C07243=1098.662,-38.451,-51.109,175.839,14.476,151.944
C07244=1098.667,-38.202,-51.121,175.841,14.477,151.943
C07245=1098.673,-37.951,-51.133,175.843,14.477,151.943
C07246=1098.679,-37.701,-51.145,175.845,14.478,151.943
C07247=1098.684,-37.452,-51.157,175.847,14.478,151.942
C07248=1098.691,-37.202,-51.169,175.849,14.479,151.942
C07249=1098.697,-36.953,-51.182,175.851,14.480,151.942
C07250=1098.702,-36.703,-51.194,175.852,14.481,151.942
C07251=1098.708,-36.453,-51.207,175.854,14.481,151.941
C07252=1098.714,-36.204,-51.219,175.856,14.482,151.941
C07253=1098.720,-35.955,-51.231,175.858,14.482,151.941
C07254=1098.726,-35.705,-51.243,175.859,14.483,151.940
C07255=1098.732,-35.455,-51.256,175.861,14.483,151.940
C07256=1098.738,-35.205,-51.269,175.863,14.484,151.940
C07257=1098.743,-34.956,-51.281,175.865,14.485,151.940
C07258=1098.749,-34.706,-51.293,175.867,14.486,151.939
C07259=1098.755,-34.456,-51.305,175.869,14.486,151.939
C07260=1098.761,-34.207,-51.317,175.871,14.487,151.939
C07261=1098.767,-33.957,-51.330,175.873,14.487,151.938
C07262=1098.773,-33.707,-51.343,175.875,14.488,151.938
C07263=1098.778,-33.458,-51.355,175.877,14.489,151.938
C07264=1098.784,-33.208,-51.367,175.879,14.490,151.938
C07265=1098.790,-32.959,-51.380,175.880,14.490,151.937
C07266=1098.797,-32.692,-51.393,175.883,14.491,151.937
C07267=1098.803,-32.424,-51.407,175.885,14.492,151.937
C07268=1098.809,-32.158,-51.419,175.887,14.493,151.936
C07269=1098.815,-31.891,-51.433,175.889,14.494,151.936
C07270=1098.821,-31.641,-51.446,175.891,14.494,151.936
C07271=1098.827,-31.391,-51.458,175.893,14.495,151.935
C07272=1098.832,-31.142,-51.471,175.895,14.495,151.935
C07273=1098.838,-30.892,-51.483,175.897,14.496,151.935
C07274=1098.845,-30.642,-51.495,175.899,14.497,151.935
C07275=1098.851,-30.392,-51.508,175.901,14.497,151.934
C07276=1098.857,-30.142,-51.520,175.903,14.498,151.934
C07277=1098.862,-29.893,-51.532,175.905,14.499,151.934
C07278=1098.868,-29.644,-51.546,175.907,14.499,151.933
C07279=1098.874,-29.394,-51.558,175.908,14.500,151.933
C07280=1098.880,-29.144,-51.571,175.911,14.500,151.933
C07281=1098.886,-28.894,-51.583,175.912,14.501,151.932
C07282=1098.891,-28.645,-51.595,175.914,14.502,151.932
C07283=1098.897,-28.395,-51.608,175.916,14.503,151.932
C07284=1098.903,-28.146,-51.621,175.918,14.503,151.932
C07285=1098.909,-27.896,-51.634,175.920,14.504,151.931
C07286=1098.916,-27.647,-51.646,175.922,14.504,151.931
C07287=1098.921,-27.397,-51.658,175.924,14.505,151.931
C07288=1098.928,-27.148,-51.671,175.926,14.506,151.930
C07289=1098.933,-26.898,-51.684,175.928,14.507,151.930
C07290=1098.939,-26.648,-51.696,175.930,14.507,151.930
C07291=1098.945,-26.398,-51.709,175.932,14.508,151.930
C07292=1098.950,-26.149,-51.722,175.934,14.509,151.929
C07293=1098.956,-25.900,-51.735,175.936,14.509,151.929
C07294=1098.962,-25.650,-51.748,175.937,14.510,151.929
C07295=1098.968,-25.400,-51.760,175.939,14.511,151.928
C07296=1098.974,-25.150,-51.773,175.942,14.511,151.928
C07297=1098.979,-24.902,-51.786,175.943,14.512,151.928
C07298=1098.985,-24.652,-51.798,175.945,14.513,151.928
C07299=1098.991,-24.402,-51.811,175.947,14.513,151.927
C07300=1098.997,-24.152,-51.824,175.949,14.514,151.927
C07301=1099.003,-23.902,-51.837,175.951,14.515,151.927
C07302=1099.008,-23.652,-51.850,175.953,14.515,151.926
C07303=1099.014,-23.404,-51.862,175.956,14.517,151.926
C07304=1099.020,-23.154,-51.875,175.958,14.517,151.926
C07305=1099.026,-22.904,-51.888,175.960,14.518,151.926
C07306=1099.032,-22.655,-51.901,175.961,14.519,151.925
C07307=1099.038,-22.405,-51.913,175.964,14.519,151.925
C07308=1099.044,-22.155,-51.926,175.965,14.520,151.925
C07309=1099.049,-21.906,-51.939,175.967,14.521,151.924
C07310=1099.055,-21.656,-51.952,175.969,14.521,151.924
C07311=1099.061,-21.406,-51.965,175.971,14.522,151.924
C07312=1099.067,-21.157,-51.978,175.973,14.522,151.923
C07313=1099.073,-20.907,-51.990,175.975,14.523,151.923
C07314=1099.079,-20.658,-52.004,175.977,14.524,151.923
C07315=1099.085,-20.408,-52.016,175.979,14.525,151.923
C07316=1099.090,-20.158,-52.029,175.981,14.525,151.922
C07317=1099.096,-19.909,-52.043,175.983,14.526,151.922
C07318=1099.102,-19.659,-52.055,175.985,14.527,151.922
C07319=1099.108,-19.410,-52.068,175.987,14.527,151.921
C07320=1099.114,-19.160,-52.081,175.989,14.528,151.921
C07321=1099.119,-18.911,-52.095,175.991,14.528,151.921
C07322=1099.125,-18.661,-52.107,175.993,14.529,151.920
C07323=1099.131,-18.412,-52.120,175.995,14.530,151.920
C07324=1099.137,-18.162,-52.133,175.997,14.531,151.920
C07325=1099.143,-17.912,-52.145,175.999,14.531,151.919
C07326=1099.149,-17.662,-52.159,176.001,14.532,151.919
C07327=1099.154,-17.412,-52.172,176.003,14.533,151.919
C07328=1099.161,-17.163,-52.185,176.005,14.534,151.919
C07329=1099.167,-16.914,-52.198,176.007,14.534,151.918
C07330=1099.173,-16.646,-52.211,176.009,14.535,151.918
C07331=1099.179,-16.378,-52.226,176.011,14.536,151.918
C07332=1099.185,-16.110,-52.240,176.014,14.536,151.917
C07333=1099.192,-15.842,-52.254,176.016,14.537,151.917
C07334=1099.198,-15.593,-52.267,176.018,14.538,151.917
C07335=1099.203,-15.343,-52.280,176.020,14.538,151.916
C07336=1099.209,-15.094,-52.294,176.022,14.539,151.916
C07337=1099.215,-14.844,-52.306,176.024,14.540,151.916
C07338=1099.221,-14.594,-52.320,176.025,14.541,151.916
C07339=1099.227,-14.344,-52.333,176.028,14.541,151.915
C07340=1099.233,-14.095,-52.346,176.030,14.542,151.915
C07341=1099.238,-13.845,-52.360,176.031,14.542,151.915
C07342=1099.244,-13.595,-52.372,176.034,14.544,151.914
C07343=1099.249,-13.347,-52.386,176.036,14.544,151.914
C07344=1099.255,-13.097,-52.398,176.038,14.545,151.914
C07345=1099.261,-12.847,-52.412,176.040,14.546,151.913
C07346=1099.267,-12.598,-52.426,176.042,14.546,151.913
C07347=1099.273,-12.348,-52.438,176.044,14.547,151.913
C07348=1099.278,-12.098,-52.452,176.046,14.547,151.912
C07349=1099.284,-11.849,-52.465,176.048,14.548,151.912
C07350=1099.290,-11.599,-52.478,176.050,14.549,151.912
C07351=1099.296,-11.350,-52.492,176.052,14.549,151.912
C07352=1099.302,-11.100,-52.505,176.054,14.550,151.911
C07353=1099.307,-10.850,-52.518,176.056,14.551,151.911
C07354=1099.313,-10.601,-52.531,176.058,14.552,151.911
C07355=1099.319,-10.351,-52.545,176.060,14.552,151.910
C07356=1099.325,-10.101,-52.558,176.062,14.553,151.910
C07357=1099.331,-9.852,-52.571,176.064,14.554,151.910
C07358=1099.336,-9.603,-52.585,176.066,14.554,151.909
C07359=1099.343,-9.353,-52.598,176.068,14.555,151.909
C07360=1099.348,-9.103,-52.611,176.070,14.556,151.909
C07361=1099.354,-8.854,-52.625,176.072,14.556,151.908
C07362=1099.359,-8.604,-52.638,176.074,14.557,151.908
C07363=1099.366,-8.355,-52.652,176.077,14.558,151.908
C07364=1099.371,-8.105,-52.665,176.079,14.559,151.908
C07365=1099.377,-7.856,-52.678,176.081,14.559,151.907
C07366=1099.383,-7.606,-52.692,176.083,14.560,151.907
C07367=1099.389,-7.357,-52.705,176.085,14.561,151.907
C07368=1099.395,-7.106,-52.718,176.087,14.561,151.906
C07369=1099.401,-6.857,-52.732,176.089,14.562,151.906
C07370=1099.407,-6.607,-52.745,176.091,14.563,151.906
C07371=1099.412,-6.358,-52.759,176.093,14.563,151.905
C07372=1099.419,-6.109,-52.772,176.095,14.564,151.905
C07373=1099.424,-5.859,-52.786,176.097,14.565,151.905
C07374=1099.430,-5.609,-52.799,176.100,14.565,151.904
C07375=1099.436,-5.360,-52.813,176.101,14.566,151.904
C07376=1099.442,-5.110,-52.826,176.104,14.566,151.904
C07377=1099.447,-4.861,-52.840,176.105,14.567,151.903
C07378=1099.453,-4.611,-52.853,176.107,14.568,151.903
C07379=1099.459,-4.362,-52.867,176.110,14.568,151.903
C07380=1099.466,-4.112,-52.881,176.111,14.569,151.902
C07381=1099.471,-3.862,-52.894,176.114,14.570,151.902
C07382=1099.476,-3.612,-52.908,176.116,14.571,151.902
C07383=1099.483,-3.363,-52.921,176.118,14.571,151.901
C07384=1099.488,-3.113,-52.935,176.120,14.572,151.901
C07385=1099.494,-2.864,-52.948,176.122,14.572,151.901
C07386=1099.500,-2.614,-52.962,176.124,14.573,151.901
C07387=1099.505,-2.365,-52.976,176.126,14.574,151.900
C07388=1099.511,-2.115,-52.990,176.128,14.574,151.900
C07389=1099.517,-1.866,-53.003,176.131,14.576,151.900
C07390=1099.522,-1.616,-53.017,176.133,14.576,151.899
C07391=1099.528,-1.367,-53.031,176.135,14.577,151.899
C07392=1099.534,-1.118,-53.044,176.137,14.577,151.899
C07393=1099.540,-0.867,-53.058,176.139,14.578,151.898
C07394=1099.546,-0.597,-53.073,176.141,14.578,151.898
C07395=1099.552,-0.328,-53.088,176.143,14.580,151.898
C07396=1099.559,-0.059,-53.102,176.146,14.580,151.897
C07397=1099.564,0.211,-53.117,176.147,14.581,151.897
C07398=1099.571,0.461,-53.131,176.150,14.582,151.897
C07399=1099.576,0.710,-53.145,176.152,14.583,151.896
C07400=1099.581,0.960,-53.158,176.154,14.583,151.896
C07401=1099.587,1.209,-53.172,176.156,14.584,151.896
C07402=1099.593,1.459,-53.186,176.158,14.584,151.895
C07403=1099.599,1.708,-53.200,176.160,14.585,151.895
C07404=1099.604,1.957,-53.214,176.162,14.585,151.895
C07405=1099.610,2.207,-53.228,176.165,14.587,151.894
C07406=1099.616,2.457,-53.242,176.167,14.588,151.894
C07407=1099.622,2.706,-53.255,176.169,14.588,151.894
C07408=1099.628,2.956,-53.269,176.171,14.589,151.893
C07409=1099.633,3.205,-53.283,176.173,14.589,151.893
C07410=1099.639,3.455,-53.297,176.175,14.590,151.893
C07411=1099.644,3.705,-53.311,176.178,14.591,151.892
C07412=1099.651,3.955,-53.324,176.180,14.591,151.892
C07413=1099.657,4.204,-53.339,176.182,14.592,151.892
C07414=1099.662,4.453,-53.353,176.184,14.592,151.891
C07415=1099.668,4.703,-53.367,176.186,14.593,151.891
C07416=1099.673,4.952,-53.381,176.188,14.594,151.891
C07417=1099.679,5.201,-53.394,176.190,14.594,151.890
C07418=1099.685,5.452,-53.408,176.192,14.596,151.890
C07419=1099.691,5.701,-53.423,176.195,14.596,151.890
C07420=1099.697,5.950,-53.437,176.196,14.597,151.889
C07421=1099.702,6.200,-53.450,176.199,14.597,151.889
C07422=1099.708,6.450,-53.465,176.201,14.598,151.889
C07423=1099.714,6.699,-53.478,176.203,14.598,151.888
C07424=1099.720,6.948,-53.493,176.205,14.599,151.888
C07425=1099.726,7.198,-53.506,176.208,14.600,151.888
C07426=1099.731,7.448,-53.520,176.209,14.601,151.887
C07427=1099.737,7.698,-53.534,176.212,14.601,151.887
C07428=1099.743,7.947,-53.549,176.214,14.602,151.887
C07429=1099.749,8.196,-53.562,176.216,14.602,151.886
C07430=1099.755,8.446,-53.576,176.218,14.603,151.886
C07431=1099.761,8.696,-53.590,176.221,14.604,151.886
C07432=1099.767,8.945,-53.605,176.222,14.604,151.885
C07433=1099.772,9.194,-53.619,176.225,14.605,151.885
C07434=1099.778,9.444,-53.633,176.226,14.605,151.885
C07435=1099.784,9.694,-53.648,176.229,14.606,151.884
C07436=1099.789,9.943,-53.662,176.231,14.607,151.884
C07437=1099.795,10.193,-53.675,176.234,14.607,151.884
C07438=1099.802,10.442,-53.690,176.235,14.608,151.883
C07439=1099.807,10.692,-53.704,176.238,14.608,151.883
C07440=1099.813,10.941,-53.717,176.239,14.609,151.883
C07441=1099.819,11.190,-53.732,176.242,14.610,151.882
C07442=1099.825,11.441,-53.746,176.244,14.611,151.882
C07443=1099.830,11.690,-53.760,176.246,14.611,151.881
C07444=1099.836,11.939,-53.775,176.248,14.612,151.881
C07445=1099.842,12.189,-53.789,176.251,14.612,151.881
C07446=1099.848,12.438,-53.804,176.253,14.613,151.880
C07447=1099.853,12.688,-53.817,176.255,14.614,151.880
C07448=1099.859,12.938,-53.832,176.258,14.614,151.880
C07449=1099.865,13.187,-53.846,176.259,14.615,151.879
C07450=1099.871,13.437,-53.860,176.262,14.615,151.879
C07451=1099.878,13.686,-53.874,176.264,14.616,151.879
C07452=1099.883,13.936,-53.888,176.266,14.617,151.878
C07453=1099.889,14.185,-53.903,176.269,14.617,151.878
C07454=1099.895,14.435,-53.917,176.271,14.618,151.878
C07455=1099.901,14.684,-53.932,176.273,14.618,151.877
C07456=1099.906,14.934,-53.946,176.275,14.619,151.877
C07457=1099.912,15.183,-53.961,176.277,14.619,151.876
C07458=1099.918,15.455,-53.976,176.280,14.620,151.876
C07459=1099.924,15.726,-53.992,176.282,14.621,151.876
C07460=1099.931,15.998,-54.008,176.285,14.622,151.875
C07461=1099.938,16.269,-54.023,176.287,14.622,151.875
C07462=1099.942,16.519,-54.038,176.289,14.623,151.875
C07463=1099.948,16.768,-54.052,176.291,14.623,151.874
C07464=1099.954,17.018,-54.067,176.294,14.624,151.874
C07465=1099.960,17.267,-54.081,176.296,14.625,151.874
C07466=1099.965,17.517,-54.095,176.298,14.625,151.873
C07467=1099.972,17.767,-54.110,176.300,14.626,151.873
C07468=1099.977,18.016,-54.124,176.303,14.627,151.872
C07469=1099.984,18.266,-54.139,176.305,14.627,151.872
C07470=1099.989,18.515,-54.154,176.307,14.628,151.872
C07471=1099.994,18.765,-54.168,176.309,14.628,151.871
C07472=1100.001,19.014,-54.183,176.311,14.629,151.871
C07473=1100.006,19.264,-54.197,176.314,14.630,151.871
C07474=1100.012,19.513,-54.211,176.316,14.630,151.870
C07475=1100.018,19.762,-54.226,176.318,14.631,151.870
C07476=1100.023,20.012,-54.241,176.320,14.632,151.869
C07477=1100.029,20.262,-54.256,176.322,14.632,151.869
C07478=1100.035,20.511,-54.270,176.325,14.633,151.869
C07479=1100.041,20.761,-54.284,176.327,14.634,151.868
C07480=1100.047,21.010,-54.299,176.329,14.634,151.868
C07481=1100.052,21.259,-54.314,176.331,14.635,151.868
C07482=1100.058,21.510,-54.328,176.334,14.636,151.867
C07483=1100.064,21.759,-54.343,176.336,14.636,151.867
C07484=1100.070,22.008,-54.358,176.338,14.637,151.867
C07485=1100.075,22.258,-54.372,176.340,14.637,151.866
C07486=1100.081,22.507,-54.387,176.342,14.638,151.866
C07487=1100.087,22.757,-54.402,176.345,14.639,151.865
C07488=1100.092,23.006,-54.417,176.347,14.639,151.865
C07489=1100.098,23.256,-54.431,176.350,14.639,151.865
C07490=1100.104,23.505,-54.446,176.351,14.640,151.864
C07491=1100.110,23.754,-54.460,176.354,14.641,151.864
C07492=1100.116,24.004,-54.476,176.357,14.641,151.863
C07493=1100.121,24.254,-54.490,176.358,14.642,151.863
C07494=1100.127,24.503,-54.505,176.361,14.642,151.863
C07495=1100.132,24.753,-54.520,176.363,14.643,151.862
C07496=1100.138,25.002,-54.535,176.365,14.644,151.862
C07497=1100.144,25.252,-54.549,176.368,14.644,151.862
C07498=1100.149,25.501,-54.564,176.370,14.645,151.861
C07499=1100.156,25.751,-54.579,176.372,14.645,151.861
C07500=1100.162,26.000,-54.593,176.375,14.646,151.861
C07501=1100.167,26.250,-54.609,176.377,14.647,151.860
C07502=1100.173,26.499,-54.624,176.379,14.647,151.860
C07503=1100.179,26.748,-54.639,176.381,14.647,151.859
C07504=1100.184,26.998,-54.653,176.384,14.649,151.859
C07505=1100.190,27.248,-54.668,176.386,14.649,151.859
C07506=1100.196,27.497,-54.683,176.388,14.649,151.858
C07507=1100.202,27.747,-54.698,176.390,14.650,151.858
C07508=1100.208,27.996,-54.713,176.393,14.650,151.857
C07509=1100.214,28.246,-54.728,176.395,14.651,151.857
C07510=1100.219,28.495,-54.743,176.398,14.652,151.857
C07511=1100.225,28.744,-54.758,176.400,14.652,151.856
C07512=1100.231,28.994,-54.773,176.403,14.653,151.856
C07513=1100.237,29.243,-54.788,176.405,14.654,151.856
C07514=1100.242,29.493,-54.802,176.407,14.654,151.855
C07515=1100.248,29.743,-54.817,176.409,14.654,151.855
C07516=1100.253,29.992,-54.832,176.412,14.655,151.854
C07517=1100.259,30.242,-54.847,176.414,14.655,151.854
C07518=1100.265,30.491,-54.863,176.416,14.656,151.854
C07519=1100.271,30.741,-54.877,176.418,14.656,151.853
C07520=1100.276,30.990,-54.893,176.421,14.657,151.853
C07521=1100.282,31.240,-54.908,176.423,14.658,151.852
C07522=1100.288,31.512,-54.925,176.425,14.658,151.852
C07523=1100.295,31.785,-54.941,176.428,14.659,151.851
C07524=1100.301,32.058,-54.957,176.431,14.659,151.851
C07525=1100.307,32.331,-54.974,176.434,14.660,151.851
C07526=1100.313,32.581,-54.989,176.436,14.660,151.850
C07527=1100.318,32.830,-55.004,176.438,14.661,151.850
C07528=1100.325,33.080,-55.019,176.440,14.662,151.849
C07529=1100.330,33.329,-55.034,176.443,14.663,151.849
C07530=1100.336,33.579,-55.049,176.445,14.663,151.849
C07531=1100.341,33.827,-55.065,176.447,14.663,151.848
C07532=1100.348,34.077,-55.080,176.450,14.664,151.848
C07533=1100.353,34.327,-55.095,176.452,14.664,151.847
C07534=1100.358,34.576,-55.111,176.455,14.665,151.847
C07535=1100.365,34.826,-55.126,176.456,14.665,151.847
C07536=1100.370,35.075,-55.141,176.459,14.666,151.846
C07537=1100.376,35.325,-55.156,176.462,14.667,151.846
C07538=1100.382,35.575,-55.171,176.464,14.667,151.845
C07539=1100.388,35.823,-55.187,176.466,14.667,151.845
C07540=1100.394,36.073,-55.202,176.469,14.668,151.844
C07541=1100.399,36.322,-55.217,176.471,14.669,151.844
C07542=1100.405,36.572,-55.232,176.473,14.669,151.844
C07543=1100.411,36.822,-55.248,176.475,14.669,151.843
C07544=1100.417,37.071,-55.262,176.478,14.670,151.843
C07545=1100.422,37.320,-55.279,176.481,14.670,151.842
C07546=1100.428,37.570,-55.294,176.483,14.671,151.842
C07547=1100.434,37.819,-55.309,176.486,14.672,151.841
C07548=1100.440,38.069,-55.324,176.488,14.672,151.841
C07549=1100.445,38.318,-55.340,176.490,14.672,151.841
C07550=1100.451,38.568,-55.355,176.492,14.673,151.840
C07551=1100.457,38.818,-55.371,176.495,14.674,151.840
C07552=1100.462,39.067,-55.386,176.497,14.674,151.840
C07553=1100.468,39.316,-55.402,176.499,14.675,151.839
C07554=1100.474,39.565,-55.417,176.502,14.676,151.839
C07555=1100.479,39.815,-55.432,176.504,14.676,151.838
C07556=1100.485,40.065,-55.448,176.507,14.676,151.838
C07557=1100.490,40.314,-55.464,176.509,14.676,151.837
C07558=1100.497,40.563,-55.479,176.512,14.677,151.837
C07559=1100.502,40.813,-55.494,176.514,14.678,151.837
C07560=1100.508,41.062,-55.510,176.516,14.678,151.836
C07561=1100.513,41.312,-55.526,176.519,14.679,151.836
C07562=1100.519,41.562,-55.541,176.521,14.679,151.835
C07563=1100.525,41.810,-55.556,176.524,14.680,151.835
C07564=1100.531,42.060,-55.572,176.526,14.680,151.834
C07565=1100.536,42.310,-55.587,176.529,14.681,151.834
C07566=1100.542,42.559,-55.603,176.531,14.681,151.834
C07567=1100.548,42.809,-55.618,176.533,14.681,151.833
C07568=1100.554,43.058,-55.635,176.536,14.682,151.833
C07569=1100.559,43.307,-55.650,176.538,14.683,151.832
C07570=1100.565,43.557,-55.665,176.541,14.683,151.832
C07571=1100.571,43.806,-55.682,176.544,14.684,151.831
C07572=1100.576,44.056,-55.697,176.546,14.684,151.831
C07573=1100.582,44.305,-55.713,176.548,14.684,151.830
C07574=1100.587,44.555,-55.729,176.550,14.684,151.830
C07575=1100.592,44.804,-55.744,176.553,14.685,151.830
C07576=1100.599,45.053,-55.759,176.555,14.686,151.829
C07577=1100.605,45.303,-55.775,176.558,14.686,151.829
C07578=1100.610,45.552,-55.791,176.561,14.687,151.828
C07579=1100.616,45.802,-55.806,176.563,14.687,151.828
C07580=1100.622,46.051,-55.823,176.565,14.688,151.827
C07581=1100.627,46.301,-55.838,176.568,14.689,151.827
C07582=1100.633,46.550,-55.854,176.570,14.689,151.827
C07583=1100.638,46.800,-55.870,176.572,14.689,151.826
C07584=1100.644,47.049,-55.886,176.575,14.690,151.826
C07585=1100.649,47.298,-55.901,176.577,14.690,151.825
C07586=1100.656,47.572,-55.919,176.580,14.691,151.825
C07587=1100.662,47.845,-55.936,176.583,14.691,151.824
C07588=1100.668,48.117,-55.953,176.586,14.692,151.824
C07589=1100.674,48.391,-55.971,176.588,14.692,151.823
C07590=1100.680,48.640,-55.987,176.591,14.692,151.823
C07591=1100.685,48.889,-56.003,176.594,14.693,151.822
C07592=1100.691,49.139,-56.018,176.596,14.694,151.822
C07593=1100.697,49.388,-56.035,176.598,14.694,151.822
C07594=1100.702,49.637,-56.050,176.601,14.695,151.821
C07595=1100.708,49.887,-56.066,176.603,14.695,151.821
C07596=1100.714,50.136,-56.082,176.605,14.695,151.820
C07597=1100.720,50.386,-56.098,176.609,14.696,151.820
C07598=1100.726,50.636,-56.114,176.611,14.696,151.819
C07599=1100.731,50.884,-56.130,176.613,14.697,151.819
C07600=1100.737,51.134,-56.146,176.616,14.698,151.818
C07601=1100.743,51.383,-56.162,176.618,14.698,151.818
C07602=1100.748,51.633,-56.179,176.621,14.698,151.817
C07603=1100.753,51.883,-56.194,176.624,14.699,151.817
C07604=1100.759,52.132,-56.210,176.626,14.699,151.817
C07605=1100.765,52.381,-56.226,176.628,14.699,151.816
C07606=1100.770,52.631,-56.242,176.631,14.700,151.815
C07607=1100.776,52.880,-56.258,176.633,14.700,151.815
C07608=1100.782,53.130,-56.274,176.636,14.700,151.815
C07609=1100.788,53.378,-56.290,176.638,14.701,151.814
C07610=1100.793,53.628,-56.306,176.641,14.701,151.814
C07611=1100.799,53.878,-56.322,176.643,14.702,151.813
C07612=1100.805,54.127,-56.338,176.645,14.702,151.813
C07613=1100.811,54.376,-56.355,176.648,14.703,151.812
C07614=1100.816,54.627,-56.371,176.651,14.703,151.812
C07615=1100.822,54.876,-56.387,176.653,14.703,151.811
C07616=1100.827,55.125,-56.403,176.656,14.704,151.811
C07617=1100.833,55.374,-56.419,176.659,14.704,151.810
C07618=1100.839,55.623,-56.435,176.661,14.704,151.810
C07619=1100.845,55.873,-56.452,176.664,14.705,151.809
C07620=1100.851,56.123,-56.467,176.666,14.705,151.809
C07621=1100.856,56.372,-56.484,176.668,14.705,151.808
C07622=1100.862,56.622,-56.500,176.671,14.706,151.808
C07623=1100.868,56.871,-56.517,176.674,14.706,151.807
C07624=1100.874,57.120,-56.533,176.676,14.706,151.807
C07625=1100.879,57.369,-56.549,176.679,14.707,151.806
C07626=1100.885,57.618,-56.565,176.681,14.707,151.806
C07627=1100.891,57.868,-56.581,176.684,14.707,151.806
C07628=1100.896,58.118,-56.597,176.687,14.708,151.805
C07629=1100.902,58.367,-56.614,176.689,14.708,151.805
C07630=1100.908,58.617,-56.630,176.692,14.708,151.804
C07631=1100.914,58.866,-56.646,176.695,14.709,151.804
C07632=1100.920,59.115,-56.662,176.697,14.709,151.803
C07633=1100.925,59.365,-56.679,176.700,14.710,151.803
C07634=1100.931,59.614,-56.695,176.702,14.710,151.802
C07635=1100.937,59.864,-56.712,176.705,14.710,151.802
C07636=1100.943,60.113,-56.728,176.708,14.711,151.801
C07637=1100.949,60.362,-56.744,176.710,14.711,151.801
C07638=1100.954,60.612,-56.761,176.712,14.711,151.800
C07639=1100.960,60.861,-56.777,176.716,14.712,151.799
C07640=1100.966,61.111,-56.794,176.718,14.712,151.799
C07641=1100.972,61.360,-56.810,176.720,14.712,151.798
C07642=1100.977,61.610,-56.827,176.723,14.713,151.798
C07643=1100.983,61.859,-56.843,176.726,14.713,151.797
C07644=1100.989,62.109,-56.859,176.728,14.713,151.797
C07645=1100.995,62.357,-56.876,176.731,14.714,151.796
C07646=1101.001,62.607,-56.893,176.734,14.714,151.796
C07647=1101.006,62.856,-56.909,176.736,14.714,151.795
C07648=1101.012,63.106,-56.926,176.739,14.715,151.795
C07649=1101.018,63.355,-56.942,176.741,14.715,151.794
C07650=1101.025,63.627,-56.960,176.745,14.715,151.794
C07651=1101.030,63.901,-56.978,176.747,14.715,151.793
C07652=1101.037,64.174,-56.996,176.750,14.716,151.793
C07653=1101.043,64.446,-57.014,176.753,14.716,151.792
C07654=1101.049,64.695,-57.030,176.756,14.716,151.792
C07655=1101.055,64.945,-57.047,176.758,14.717,151.791
C07656=1101.061,65.194,-57.064,176.761,14.716,151.791
C07657=1101.066,65.443,-57.081,176.764,14.717,151.790
C07658=1101.072,65.693,-57.097,176.766,14.717,151.790
C07659=1101.078,65.942,-57.114,176.769,14.717,151.789
C07660=1101.083,66.192,-57.130,176.772,14.718,151.789
C07661=1101.089,66.441,-57.147,176.774,14.718,151.788
C07662=1101.095,66.690,-57.164,176.776,14.718,151.788
C07663=1101.101,66.939,-57.181,176.780,14.719,151.787
C07664=1101.106,67.189,-57.197,176.782,14.719,151.786
C07665=1101.112,67.438,-57.214,176.785,14.720,151.786
C07666=1101.117,67.688,-57.231,176.788,14.719,151.785
C07667=1101.124,67.937,-57.248,176.790,14.720,151.785
C07668=1101.129,68.187,-57.265,176.793,14.720,151.784
C07669=1101.135,68.436,-57.281,176.796,14.720,151.784
C07670=1101.141,68.686,-57.299,176.798,14.720,151.783
C07671=1101.146,68.935,-57.315,176.801,14.721,151.783
C07672=1101.152,69.185,-57.332,176.804,14.721,151.782
C07673=1101.158,69.433,-57.349,176.806,14.722,151.782
C07674=1101.163,69.683,-57.365,176.809,14.722,151.781
C07675=1101.169,69.932,-57.382,176.812,14.721,151.781
C07676=1101.174,70.182,-57.399,176.814,14.722,151.780
C07677=1101.181,70.431,-57.416,176.817,14.722,151.780
C07678=1101.186,70.680,-57.432,176.819,14.722,151.779
C07679=1101.191,70.929,-57.450,176.822,14.723,151.779
C07680=1101.197,71.179,-57.466,176.825,14.723,151.778
C07681=1101.203,71.429,-57.483,176.828,14.724,151.777
C07682=1101.209,71.678,-57.500,176.830,14.724,151.777
C07683=1101.215,71.927,-57.517,176.833,14.724,151.776
C07684=1101.220,72.176,-57.535,176.836,14.724,151.776
C07685=1101.226,72.426,-57.551,176.838,14.725,151.775
C07686=1101.231,72.675,-57.568,176.841,14.724,151.775
C07687=1101.237,72.925,-57.586,176.844,14.725,151.774
C07688=1101.243,73.174,-57.602,176.847,14.725,151.774
C07689=1101.248,73.423,-57.619,176.850,14.726,151.773
C07690=1101.255,73.673,-57.636,176.852,14.726,151.773
C07691=1101.260,73.922,-57.654,176.855,14.725,151.772
C07692=1101.265,74.172,-57.670,176.858,14.726,151.771
C07693=1101.272,74.420,-57.687,176.860,14.726,151.771
C07694=1101.277,74.670,-57.704,176.863,14.726,151.770
C07695=1101.282,74.919,-57.722,176.866,14.727,151.770
C07696=1101.288,75.169,-57.739,176.868,14.727,151.769
C07697=1101.295,75.418,-57.756,176.872,14.727,151.769
C07698=1101.300,75.668,-57.773,176.874,14.727,151.768
C07699=1101.305,75.917,-57.790,176.876,14.727,151.768
C07700=1101.311,76.166,-57.807,176.880,14.728,151.767
C07701=1101.317,76.415,-57.824,176.882,14.728,151.766
C07702=1101.322,76.665,-57.841,176.885,14.728,151.766
C07703=1101.329,76.914,-57.858,176.888,14.728,151.765
C07704=1101.334,77.163,-57.876,176.890,14.728,151.765
C07705=1101.340,77.413,-57.893,176.893,14.729,151.764
C07706=1101.345,77.662,-57.910,176.896,14.729,151.764
C07707=1101.351,77.911,-57.927,176.898,14.729,151.763
C07708=1101.357,78.161,-57.945,176.902,14.729,151.762
C07709=1101.363,78.410,-57.962,176.904,14.729,151.762
C07710=1101.368,78.660,-57.979,176.907,14.730,151.761
C07711=1101.373,78.909,-57.997,176.910,14.729,151.761
C07712=1101.380,79.158,-58.014,176.912,14.729,151.760
C07713=1101.385,79.408,-58.031,176.916,14.730,151.760
C07714=1101.391,79.680,-58.050,176.918,14.730,151.759
C07715=1101.397,79.953,-58.069,176.922,14.730,151.758
C07716=1101.404,80.226,-58.089,176.925,14.731,151.758
C07717=1101.410,80.499,-58.107,176.927,14.731,151.757
C07718=1101.416,80.747,-58.124,176.931,14.731,151.757
C07719=1101.421,80.997,-58.141,176.933,14.731,151.756
C07720=1101.427,81.246,-58.159,176.936,14.731,151.755
C07721=1101.432,81.495,-58.176,176.939,14.731,151.755
C07722=1101.438,81.745,-58.194,176.941,14.731,151.754
C07723=1101.444,81.995,-58.211,176.945,14.732,151.754
C07724=1101.449,82.244,-58.229,176.947,14.732,151.753
C07725=1101.455,82.493,-58.246,176.950,14.732,151.752
C07726=1101.461,82.742,-58.264,176.953,14.732,151.752
C07727=1101.466,82.991,-58.282,176.955,14.732,151.751
C07728=1101.472,83.241,-58.299,176.959,14.732,151.751
C07729=1101.477,83.490,-58.316,176.961,14.732,151.750
C07730=1101.483,83.740,-58.334,176.965,14.733,151.750
C07731=1101.489,83.989,-58.352,176.967,14.733,151.749
C07732=1101.494,84.238,-58.369,176.970,14.733,151.748
C07733=1101.500,84.488,-58.387,176.973,14.733,151.748
C07734=1101.506,84.737,-58.403,176.975,14.733,151.747
C07735=1101.512,84.986,-58.421,176.979,14.733,151.747
C07736=1101.517,85.235,-58.439,176.981,14.733,151.746
C07737=1101.523,85.485,-58.457,176.984,14.733,151.745
C07738=1101.529,85.734,-58.474,176.987,14.734,151.745
C07739=1101.534,85.983,-58.492,176.989,14.734,151.744
C07740=1101.541,86.233,-58.510,176.993,14.734,151.744
C07741=1101.546,86.482,-58.527,176.995,14.734,151.743
C07742=1101.552,86.731,-58.545,176.998,14.733,151.742
C07743=1101.558,86.980,-58.563,177.001,14.734,151.742
C07744=1101.563,87.230,-58.580,177.004,14.734,151.741
C07745=1101.569,87.479,-58.598,177.007,14.734,151.741
C07746=1101.575,87.728,-58.616,177.010,14.734,151.740
C07747=1101.580,87.978,-58.634,177.012,14.734,151.739
C07748=1101.586,88.227,-58.652,177.016,14.734,151.739
C07749=1101.591,88.476,-58.669,177.018,14.734,151.738
C07750=1101.597,88.725,-58.687,177.021,14.735,151.737
C07751=1101.603,88.975,-58.705,177.024,14.734,151.737
C07752=1101.608,89.224,-58.722,177.026,14.734,151.736
C07753=1101.615,89.474,-58.740,177.030,14.734,151.736
C07754=1101.620,89.723,-58.758,177.033,14.734,151.735
C07755=1101.626,89.972,-58.776,177.036,14.735,151.734
C07756=1101.632,90.222,-58.793,177.038,14.735,151.734
C07757=1101.637,90.471,-58.811,177.042,14.735,151.733
C07758=1101.643,90.721,-58.829,177.044,14.735,151.732
C07759=1101.649,90.970,-58.847,177.047,14.735,151.732
C07760=1101.655,91.218,-58.865,177.050,14.735,151.731
C07761=1101.660,91.468,-58.883,177.053,14.734,151.731
C07762=1101.666,91.717,-58.901,177.056,14.735,151.730
C07763=1101.672,91.967,-58.919,177.059,14.735,151.729
C07764=1101.677,92.216,-58.936,177.061,14.735,151.729
C07765=1101.682,92.465,-58.955,177.065,14.735,151.728
C07766=1101.688,92.715,-58.973,177.067,14.735,151.727
C07767=1101.694,92.963,-58.991,177.071,14.735,151.727
C07768=1101.700,93.213,-59.009,177.073,14.735,151.726
C07769=1101.706,93.462,-59.026,177.077,14.735,151.726
C07770=1101.710,93.712,-59.044,177.079,14.735,151.725
C07771=1101.717,93.961,-59.062,177.082,14.735,151.724
C07772=1101.722,94.210,-59.081,177.085,14.736,151.724
C07773=1101.728,94.460,-59.099,177.088,14.735,151.723
C07774=1101.733,94.709,-59.117,177.091,14.736,151.722
C07775=1101.739,94.959,-59.135,177.094,14.735,151.722
C07776=1101.745,95.207,-59.153,177.097,14.735,151.721
C07777=1101.750,95.456,-59.171,177.100,14.735,151.721
C07778=1101.757,95.730,-59.191,177.103,14.735,151.720
C07779=1101.763,96.002,-59.211,177.106,14.735,151.719
C07780=1101.769,96.275,-59.231,177.109,14.735,151.718
C07781=1101.775,96.547,-59.251,177.113,14.735,151.718
C07782=1101.781,96.797,-59.268,177.116,14.735,151.717
C07783=1101.787,97.046,-59.287,177.118,14.735,151.716
C07784=1101.792,97.295,-59.305,177.122,14.735,151.716
C07785=1101.798,97.545,-59.323,177.124,14.735,151.715
C07786=1101.803,97.793,-59.342,177.128,14.735,151.714
C07787=1101.809,98.043,-59.360,177.130,14.735,151.714
C07788=1101.815,98.292,-59.377,177.134,14.735,151.713
C07789=1101.821,98.542,-59.397,177.136,14.735,151.712
C07790=1101.826,98.791,-59.414,177.140,14.735,151.712
C07791=1101.833,99.040,-59.433,177.142,14.735,151.711
C07792=1101.837,99.289,-59.451,177.145,14.735,151.710
C07793=1101.844,99.539,-59.469,177.149,14.735,151.710
C07794=1101.850,99.788,-59.488,177.151,14.735,151.709
C07795=1101.855,100.037,-59.506,177.155,14.735,151.708
C07796=1101.861,100.287,-59.524,177.157,14.735,151.708
C07797=1101.867,100.536,-59.542,177.161,14.735,151.707
C07798=1101.872,100.785,-59.561,177.164,14.734,151.706
C07799=1101.878,101.034,-59.579,177.166,14.734,151.706
C07800=1101.884,101.283,-59.598,177.170,14.734,151.705
C07801=1101.889,101.533,-59.616,177.172,14.734,151.704
C07802=1101.895,101.782,-59.635,177.176,14.734,151.704
C07803=1101.901,102.032,-59.653,177.179,14.734,151.703
C07804=1101.906,102.280,-59.672,177.182,14.734,151.702
C07805=1101.912,102.530,-59.690,177.185,14.734,151.702
C07806=1101.917,102.779,-59.708,177.187,14.734,151.701
C07807=1101.924,103.028,-59.727,177.191,14.734,151.700
C07808=1101.928,103.277,-59.745,177.193,14.734,151.700
C07809=1101.935,103.526,-59.764,177.197,14.734,151.699
C07810=1101.940,103.776,-59.782,177.200,14.733,151.698
C07811=1101.945,104.025,-59.801,177.203,14.734,151.698
C07812=1101.951,104.275,-59.819,177.206,14.733,151.697
C07813=1101.957,104.524,-59.838,177.209,14.734,151.696
C07814=1101.963,104.773,-59.857,177.212,14.733,151.696
C07815=1101.968,105.022,-59.875,177.215,14.733,151.695
C07816=1101.974,105.271,-59.894,177.218,14.733,151.694
C07817=1101.980,105.521,-59.913,177.221,14.733,151.693
C07818=1101.985,105.770,-59.931,177.224,14.733,151.693
C07819=1101.991,106.019,-59.950,177.227,14.733,151.692
C07820=1101.997,106.269,-59.969,177.231,14.733,151.691
C07821=1102.002,106.518,-59.986,177.233,14.732,151.691
C07822=1102.008,106.767,-60.006,177.237,14.733,151.690
C07823=1102.013,107.016,-60.024,177.239,14.732,151.689
C07824=1102.019,107.265,-60.043,177.243,14.732,151.689
C07825=1102.025,107.515,-60.062,177.246,14.732,151.688
C07826=1102.031,107.763,-60.080,177.248,14.732,151.687
C07827=1102.036,108.013,-60.099,177.252,14.732,151.686
C07828=1102.042,108.262,-60.118,177.255,14.731,151.686
C07829=1102.048,108.511,-60.136,177.258,14.732,151.685
C07830=1102.053,108.761,-60.155,177.261,14.731,151.684
C07831=1102.059,109.010,-60.174,177.264,14.731,151.684
C07832=1102.065,109.259,-60.193,177.267,14.731,151.683
C07833=1102.070,109.508,-60.212,177.271,14.731,151.682
C07834=1102.076,109.758,-60.231,177.273,14.731,151.682
C07835=1102.082,110.007,-60.249,177.276,14.730,151.681
C07836=1102.087,110.256,-60.268,177.280,14.730,151.680
C07837=1102.093,110.505,-60.287,177.283,14.730,151.679
C07838=1102.099,110.755,-60.306,177.286,14.730,151.679
C07839=1102.105,111.004,-60.325,177.289,14.729,151.678
C07840=1102.110,111.253,-60.344,177.292,14.730,151.677
C07841=1102.117,111.502,-60.363,177.295,14.729,151.676
C07842=1102.122,111.775,-60.383,177.299,14.729,151.676
C07843=1102.129,112.048,-60.404,177.303,14.729,151.675
C07844=1102.135,112.320,-60.424,177.305,14.729,151.674
C07845=1102.141,112.593,-60.446,177.309,14.729,151.673
C07846=1102.147,112.843,-60.465,177.312,14.728,151.673
C07847=1102.152,113.092,-60.484,177.315,14.728,151.672
C07848=1102.158,113.341,-60.503,177.318,14.728,151.671
C07849=1102.164,113.590,-60.522,177.322,14.728,151.670
C07850=1102.170,113.840,-60.541,177.325,14.727,151.670
C07851=1102.175,114.088,-60.560,177.328,14.727,151.669
C07852=1102.180,114.338,-60.579,177.331,14.727,151.668
C07853=1102.187,114.587,-60.598,177.334,14.727,151.667
C07854=1102.193,114.836,-60.617,177.337,14.727,151.667
C07855=1102.198,115.085,-60.636,177.341,14.727,151.666
C07856=1102.203,115.334,-60.655,177.344,14.726,151.665
C07857=1102.209,115.584,-60.674,177.346,14.726,151.664
C07858=1102.214,115.833,-60.693,177.350,14.726,151.664
C07859=1102.220,116.082,-60.713,177.353,14.725,151.663
C07860=1102.225,116.331,-60.732,177.356,14.725,151.662
C07861=1102.231,116.581,-60.751,177.359,14.725,151.661
C07862=1102.237,116.829,-60.771,177.363,14.725,151.661
C07863=1102.242,117.078,-60.790,177.366,14.724,151.660
C07864=1102.248,117.328,-60.809,177.369,14.725,151.659
C07865=1102.254,117.577,-60.828,177.372,14.724,151.659
C07866=1102.259,117.827,-60.848,177.376,14.724,151.658
C07867=1102.264,118.075,-60.866,177.378,14.724,151.657
C07868=1102.270,118.325,-60.886,177.382,14.724,151.656
C07869=1102.276,118.574,-60.905,177.385,14.723,151.656
C07870=1102.282,118.823,-60.925,177.389,14.723,151.655
C07871=1102.287,119.073,-60.944,177.391,14.723,151.654
C07872=1102.293,119.321,-60.963,177.395,14.723,151.653
C07873=1102.298,119.571,-60.982,177.398,14.722,151.653
C07874=1102.304,119.820,-61.002,177.401,14.722,151.652
C07875=1102.310,120.069,-61.021,177.404,14.722,151.651
C07876=1102.316,120.318,-61.041,177.407,14.721,151.650
C07877=1102.321,120.568,-61.060,177.411,14.722,151.650
C07878=1102.327,120.816,-61.080,177.413,14.721,151.649
C07879=1102.332,121.066,-61.099,177.417,14.721,151.648
C07880=1102.337,121.315,-61.119,177.420,14.721,151.647
C07881=1102.343,121.565,-61.138,177.423,14.721,151.647
C07882=1102.349,121.813,-61.158,177.427,14.720,151.646
C07883=1102.355,122.063,-61.177,177.430,14.720,151.645
C07884=1102.360,122.312,-61.196,177.433,14.719,151.644
C07885=1102.366,122.560,-61.216,177.437,14.719,151.643
C07886=1102.371,122.810,-61.235,177.439,14.719,151.643
C07887=1102.377,123.059,-61.254,177.443,14.719,151.642
C07888=1102.383,123.308,-61.274,177.446,14.718,151.641
C07889=1102.389,123.557,-61.294,177.450,14.718,151.640
C07890=1102.394,123.807,-61.314,177.453,14.718,151.639
C07891=1102.400,124.056,-61.333,177.456,14.718,151.639
C07892=1102.405,124.305,-61.353,177.459,14.717,151.638
C07893=1102.411,124.554,-61.373,177.462,14.716,151.637
C07894=1102.417,124.804,-61.392,177.466,14.716,151.636
C07895=1102.423,125.053,-61.412,177.469,14.716,151.636
C07896=1102.429,125.302,-61.431,177.472,14.715,151.635
C07897=1102.434,125.551,-61.452,177.475,14.715,151.634
C07898=1102.440,125.801,-61.471,177.479,14.715,151.633
C07899=1102.446,126.049,-61.491,177.482,14.714,151.632
C07900=1102.451,126.299,-61.510,177.486,14.714,151.632
C07901=1102.457,126.547,-61.530,177.488,14.714,151.631
C07902=1102.463,126.796,-61.549,177.492,14.713,151.630
C07903=1102.468,127.045,-61.569,177.495,14.713,151.629
C07904=1102.473,127.295,-61.589,177.499,14.713,151.628
C07905=1102.479,127.544,-61.609,177.502,14.712,151.627
C07906=1102.486,127.817,-61.630,177.505,14.712,151.627
C07907=1102.492,128.090,-61.652,177.509,14.712,151.626
C07908=1102.499,128.362,-61.674,177.513,14.711,151.625
C07909=1102.505,128.635,-61.695,177.516,14.711,151.624
C07910=1102.511,128.885,-61.714,177.519,14.710,151.623
C07911=1102.516,129.134,-61.735,177.523,14.710,151.622
C07912=1102.522,129.382,-61.755,177.526,14.709,151.622
C07913=1102.528,129.632,-61.774,177.530,14.709,151.621
C07914=1102.534,129.881,-61.794,177.533,14.708,151.620
C07915=1102.539,130.130,-61.815,177.537,14.708,151.619
C07916=1102.545,130.379,-61.834,177.539,14.707,151.618
C07917=1102.551,130.628,-61.854,177.543,14.707,151.617
C07918=1102.557,130.877,-61.874,177.546,14.707,151.617
C07919=1102.562,131.127,-61.894,177.550,14.706,151.616
C07920=1102.568,131.375,-61.914,177.553,14.706,151.615
C07921=1102.574,131.624,-61.934,177.557,14.705,151.614
C07922=1102.580,131.873,-61.954,177.560,14.705,151.613
C07923=1102.585,132.124,-61.974,177.564,14.705,151.612
C07924=1102.591,132.372,-61.994,177.566,14.704,151.612
C07925=1102.597,132.621,-62.014,177.570,14.704,151.611
C07926=1102.603,132.870,-62.034,177.573,14.703,151.610
C07927=1102.608,133.120,-62.053,177.577,14.703,151.609
C07928=1102.613,133.369,-62.074,177.580,14.702,151.608
C07929=1102.619,133.618,-62.094,177.584,14.702,151.607
C07930=1102.625,133.867,-62.115,177.587,14.702,151.607
C07931=1102.631,134.116,-62.135,177.591,14.701,151.606
C07932=1102.636,134.365,-62.154,177.593,14.701,151.605
C07933=1102.642,134.614,-62.174,177.597,14.701,151.604
C07934=1102.647,134.863,-62.195,177.600,14.700,151.603
C07935=1102.653,135.112,-62.215,177.604,14.700,151.602
C07936=1102.659,135.362,-62.235,177.607,14.699,151.602
C07937=1102.665,135.611,-62.256,177.611,14.699,151.601
C07938=1102.670,135.860,-62.275,177.614,14.698,151.600
C07939=1102.676,136.109,-62.295,177.617,14.698,151.599
C07940=1102.682,136.358,-62.315,177.621,14.697,151.598
C07941=1102.687,136.607,-62.336,177.624,14.697,151.597
C07942=1102.693,136.856,-62.356,177.627,14.696,151.597
C07943=1102.698,137.105,-62.377,177.631,14.696,151.596
C07944=1102.705,137.355,-62.397,177.634,14.695,151.595
C07945=1102.710,137.604,-62.417,177.638,14.695,151.594
C07946=1102.715,137.853,-62.438,177.641,14.694,151.593
C07947=1102.721,138.102,-62.458,177.644,14.693,151.592
C07948=1102.727,138.351,-62.478,177.648,14.693,151.591
C07949=1102.733,138.600,-62.498,177.651,14.692,151.591
C07950=1102.738,138.849,-62.519,177.655,14.692,151.590
C07951=1102.744,139.098,-62.539,177.658,14.692,151.589
C07952=1102.750,139.347,-62.560,177.662,14.691,151.588
C07953=1102.755,139.597,-62.580,177.665,14.690,151.587
C07954=1102.761,139.845,-62.600,177.669,14.690,151.586
C07955=1102.766,140.094,-62.621,177.672,14.690,151.585
C07956=1102.773,140.344,-62.641,177.675,14.689,151.585
C07957=1102.778,140.593,-62.662,177.679,14.688,151.584
C07958=1102.783,140.842,-62.682,177.682,14.688,151.583
C07959=1102.789,141.091,-62.702,177.685,14.688,151.582
C07960=1102.795,141.340,-62.724,177.689,14.687,151.581
C07961=1102.801,141.589,-62.745,177.692,14.686,151.580
C07962=1102.807,141.838,-62.764,177.696,14.686,151.579
C07963=1102.812,142.087,-62.785,177.699,14.686,151.578
C07964=1102.817,142.336,-62.806,177.703,14.685,151.578
C07965=1102.822,142.586,-62.826,177.706,14.684,151.577
C07966=1102.829,142.835,-62.846,177.710,14.684,151.576
C07967=1102.835,143.084,-62.868,177.713,14.684,151.575
C07968=1102.840,143.333,-62.888,177.717,14.683,151.574
C07969=1102.846,143.582,-62.908,177.720,14.682,151.573
C07970=1102.852,143.854,-62.931,177.724,14.682,151.572
C07971=1102.858,144.127,-62.953,177.728,14.681,151.571
C07972=1102.864,144.399,-62.976,177.732,14.681,151.570
C07973=1102.870,144.672,-62.999,177.735,14.680,151.569
C07974=1102.877,144.921,-63.020,177.739,14.680,151.568
C07975=1102.882,145.170,-63.041,177.742,14.679,151.568
C07976=1102.888,145.419,-63.061,177.746,14.679,151.567
C07977=1102.893,145.668,-63.081,177.749,14.678,151.566
C07978=1102.899,145.917,-63.103,177.753,14.677,151.565
C07979=1102.904,146.167,-63.124,177.756,14.676,151.564
C07980=1102.910,146.416,-63.144,177.760,14.676,151.563
C07981=1102.917,146.665,-63.165,177.763,14.675,151.562
C07982=1102.922,146.914,-63.186,177.767,14.675,151.561
C07983=1102.927,147.163,-63.206,177.770,14.674,151.560
C07984=1102.933,147.412,-63.228,177.774,14.674,151.559
C07985=1102.939,147.661,-63.248,177.777,14.673,151.558
C07986=1102.945,147.909,-63.269,177.781,14.672,151.558
C07987=1102.951,148.159,-63.290,177.785,14.671,151.557
C07988=1102.956,148.408,-63.311,177.788,14.671,151.556
C07989=1102.961,148.657,-63.332,177.792,14.671,151.555
C07990=1102.967,148.907,-63.353,177.795,14.670,151.554
C07991=1102.973,149.155,-63.374,177.799,14.670,151.553
C07992=1102.978,149.404,-63.395,177.803,14.669,151.552
C07993=1102.984,149.653,-63.416,177.806,14.669,151.551
C07994=1102.990,149.903,-63.437,177.810,14.668,151.550
C07995=1102.995,150.151,-63.458,177.813,14.667,151.549
C07996=1103.001,150.401,-63.479,177.817,14.666,151.548
C07997=1103.007,150.649,-63.500,177.821,14.666,151.548
C07998=1103.013,150.898,-63.520,177.824,14.665,151.547
C07999=1103.019,151.147,-63.542,177.828,14.665,151.546
C08000=1103.024,151.397,-63.562,177.831,14.664,151.545
C08001=1103.030,151.646,-63.584,177.835,14.664,151.544
C08002=1103.035,151.895,-63.605,177.838,14.663,151.543
C08003=1103.041,152.143,-63.626,177.842,14.662,151.542
C08004=1103.047,152.393,-63.647,177.845,14.661,151.541
C08005=1103.052,152.642,-63.668,177.849,14.661,151.540
C08006=1103.059,152.891,-63.690,177.852,14.660,151.539
C08007=1103.063,153.140,-63.711,177.856,14.660,151.538
C08008=1103.069,153.389,-63.732,177.859,14.659,151.537
C08009=1103.075,153.638,-63.754,177.863,14.658,151.537
C08010=1103.080,153.887,-63.774,177.866,14.658,151.536
C08011=1103.086,154.136,-63.796,177.871,14.657,151.535
C08012=1103.092,154.385,-63.817,177.874,14.656,151.534
C08013=1103.097,154.634,-63.838,177.878,14.656,151.533
C08014=1103.103,154.883,-63.859,177.881,14.655,151.532
C08015=1103.109,155.132,-63.881,177.885,14.654,151.531
C08016=1103.115,155.382,-63.902,177.888,14.653,151.530
C08017=1103.120,155.630,-63.923,177.892,14.653,151.529
C08018=1103.126,155.879,-63.945,177.895,14.652,151.528
C08019=1103.132,156.128,-63.965,177.899,14.652,151.527
C08020=1103.137,156.378,-63.987,177.903,14.650,151.526
C08021=1103.143,156.626,-64.009,177.906,14.650,151.525
C08022=1103.149,156.876,-64.030,177.910,14.649,151.524
C08023=1103.154,157.124,-64.051,177.914,14.649,151.523
C08024=1103.160,157.374,-64.072,177.918,14.648,151.522
C08025=1103.166,157.622,-64.094,177.921,14.647,151.521
C08026=1103.171,157.871,-64.116,177.925,14.647,151.520
C08027=1103.177,158.120,-64.137,177.928,14.646,151.520
C08028=1103.182,158.369,-64.158,177.932,14.645,151.518
C08029=1103.188,158.619,-64.179,177.935,14.644,151.518
C08030=1103.194,158.868,-64.201,177.939,14.644,151.517
C08031=1103.199,159.117,-64.223,177.943,14.643,151.516
C08032=1103.205,159.366,-64.244,177.947,14.643,151.515
C08033=1103.211,159.615,-64.266,177.950,14.642,151.514
C08034=1103.217,159.887,-64.289,177.954,14.641,151.513
C08035=1103.223,160.159,-64.313,177.958,14.640,151.512
C08036=1103.230,160.432,-64.337,177.962,14.639,151.511
C08037=1103.236,160.704,-64.360,177.966,14.638,151.509
C08038=1103.241,160.952,-64.382,177.970,14.638,151.509
C08039=1103.247,161.202,-64.404,177.973,14.637,151.508
C08040=1103.253,161.450,-64.425,177.977,14.636,151.507
C08041=1103.258,161.700,-64.447,177.981,14.635,151.506
C08042=1103.264,161.948,-64.468,177.985,14.635,151.505
C08043=1103.270,162.197,-64.490,177.988,14.634,151.504
C08044=1103.275,162.446,-64.512,177.992,14.633,151.503
C08045=1103.281,162.695,-64.533,177.995,14.632,151.502
C08046=1103.286,162.944,-64.555,177.999,14.632,151.501
C08047=1103.292,163.193,-64.577,178.003,14.631,151.500
C08048=1103.298,163.443,-64.599,178.006,14.630,151.499
C08049=1103.303,163.691,-64.620,178.010,14.630,151.498
C08050=1103.309,163.941,-64.643,178.014,14.629,151.497
C08051=1103.314,164.189,-64.664,178.018,14.629,151.496
C08052=1103.319,164.439,-64.686,178.021,14.627,151.495
C08053=1103.325,164.687,-64.707,178.025,14.627,151.494
C08054=1103.330,164.937,-64.730,178.028,14.626,151.493
C08055=1103.336,165.185,-64.751,178.032,14.625,151.492
C08056=1103.341,165.435,-64.773,178.036,14.625,151.491
C08057=1103.347,165.683,-64.795,178.040,14.624,151.490
C08058=1103.353,165.932,-64.817,178.043,14.623,151.489
C08059=1103.359,166.182,-64.839,178.047,14.622,151.488
C08060=1103.364,166.430,-64.861,178.051,14.622,151.487
C08061=1103.370,166.680,-64.883,178.055,14.621,151.486
C08062=1103.375,166.928,-64.904,178.059,14.621,151.485
C08063=1103.381,167.177,-64.927,178.062,14.619,151.484
C08064=1103.387,167.426,-64.949,178.066,14.619,151.483
C08065=1103.392,167.675,-64.970,178.069,14.618,151.482
C08066=1103.398,167.925,-64.992,178.073,14.617,151.481
C08067=1103.403,168.173,-65.015,178.077,14.616,151.480
C08068=1103.409,168.422,-65.037,178.081,14.616,151.479
C08069=1103.414,168.671,-65.059,178.084,14.615,151.478
C08070=1103.421,168.920,-65.081,178.088,14.614,151.477
C08071=1103.426,169.169,-65.103,178.091,14.613,151.476
C08072=1103.432,169.418,-65.125,178.096,14.612,151.475
C08073=1103.437,169.668,-65.147,178.100,14.612,151.474
C08074=1103.442,169.916,-65.170,178.103,14.611,151.473
C08075=1103.449,170.165,-65.191,178.107,14.610,151.472
C08076=1103.454,170.414,-65.214,178.110,14.609,151.471
C08077=1103.459,170.663,-65.236,178.115,14.608,151.470
C08078=1103.465,170.912,-65.258,178.118,14.607,151.469
C08079=1103.471,171.161,-65.281,178.122,14.607,151.468
C08080=1103.477,171.409,-65.302,178.126,14.606,151.467
C08081=1103.482,171.658,-65.325,178.130,14.605,151.466
C08082=1103.488,171.908,-65.347,178.133,14.604,151.465
C08083=1103.494,172.157,-65.369,178.137,14.603,151.464
C08084=1103.499,172.405,-65.391,178.141,14.602,151.463
C08085=1103.504,172.655,-65.413,178.145,14.602,151.462
C08086=1103.511,172.903,-65.436,178.149,14.601,151.461
C08087=1103.516,173.153,-65.458,178.152,14.600,151.460
C08088=1103.521,173.401,-65.481,178.156,14.599,151.459
C08089=1103.528,173.650,-65.502,178.160,14.598,151.458
C08090=1103.533,173.899,-65.525,178.164,14.598,151.457
C08091=1103.539,174.149,-65.547,178.167,14.596,151.456
C08092=1103.545,174.396,-65.569,178.172,14.596,151.455
C08093=1103.550,174.646,-65.592,178.175,14.594,151.454
C08094=1103.556,174.895,-65.615,178.179,14.594,151.453
C08095=1103.561,175.144,-65.638,178.182,14.593,151.452
C08096=1103.568,175.393,-65.659,178.187,14.592,151.451
C08097=1103.573,175.641,-65.682,178.190,14.591,151.450
C08098=1103.579,175.913,-65.707,178.194,14.590,151.449
C08099=1103.585,176.185,-65.731,178.199,14.589,151.447
C08100=1103.592,176.457,-65.755,178.203,14.589,151.446
C08101=1103.598,176.729,-65.779,178.207,14.588,151.445
C08102=1103.604,176.978,-65.802,178.211,14.587,151.444
C08103=1103.609,177.227,-65.825,178.215,14.586,151.443
C08104=1103.615,177.476,-65.848,178.219,14.585,151.442
C08105=1103.621,177.725,-65.870,178.223,14.584,151.441
C08106=1103.627,177.974,-65.893,178.226,14.583,151.440
C08107=1103.632,178.223,-65.915,178.230,14.582,151.439
C08108=1103.637,178.471,-65.938,178.234,14.581,151.438
C08109=1103.643,178.720,-65.961,178.238,14.580,151.437
C08110=1103.650,178.969,-65.983,178.242,14.579,151.436
C08111=1103.655,179.218,-66.005,178.246,14.578,151.434
C08112=1103.661,179.467,-66.028,178.249,14.577,151.433
C08113=1103.667,179.716,-66.051,178.254,14.576,151.432
C08114=1103.672,179.965,-66.074,178.258,14.576,151.431
C08115=1103.679,180.214,-66.096,178.261,14.574,151.430
C08116=1103.684,180.463,-66.119,178.266,14.574,151.429
C08117=1103.690,180.712,-66.142,178.269,14.572,151.428
C08118=1103.696,180.961,-66.164,178.273,14.572,151.427
C08119=1103.701,181.210,-66.187,178.277,14.570,151.426
C08120=1103.707,181.459,-66.210,178.281,14.570,151.425
C08121=1103.713,181.707,-66.232,178.284,14.568,151.424
C08122=1103.719,181.956,-66.255,178.289,14.568,151.423
C08123=1103.724,182.204,-66.278,178.292,14.567,151.422
C08124=1103.730,182.453,-66.301,178.296,14.566,151.421
C08125=1103.736,182.703,-66.323,178.300,14.565,151.420
C08126=1103.741,182.952,-66.346,178.304,14.564,151.418
C08127=1103.747,183.201,-66.369,178.309,14.563,151.417
C08128=1103.753,183.450,-66.392,178.312,14.562,151.416
C08129=1103.759,183.698,-66.415,178.316,14.561,151.415
C08130=1103.765,183.947,-66.438,178.320,14.560,151.414
C08131=1103.771,184.196,-66.460,178.324,14.559,151.413
C08132=1103.776,184.445,-66.483,178.327,14.558,151.412
C08133=1103.782,184.694,-66.506,178.332,14.557,151.411
C08134=1103.788,184.943,-66.530,178.336,14.555,151.410
C08135=1103.794,185.192,-66.553,178.340,14.555,151.409
C08136=1103.800,185.440,-66.576,178.343,14.553,151.407
C08137=1103.805,185.689,-66.599,178.347,14.553,151.406
C08138=1103.810,185.938,-66.622,178.352,14.552,151.405
C08139=1103.816,186.187,-66.645,178.355,14.551,151.404
C08140=1103.822,186.436,-66.668,178.359,14.550,151.403
C08141=1103.828,186.685,-66.691,178.363,14.549,151.402
C08142=1103.833,186.933,-66.714,178.367,14.548,151.401
C08143=1103.838,187.183,-66.738,178.371,14.547,151.400
C08144=1103.844,187.432,-66.761,178.375,14.547,151.399
C08145=1103.850,187.680,-66.784,178.379,14.545,151.398
C08146=1103.855,187.929,-66.807,178.383,14.544,151.397
C08147=1103.862,188.178,-66.830,178.387,14.544,151.396
C08148=1103.867,188.427,-66.854,178.391,14.542,151.395
C08149=1103.872,188.676,-66.877,178.395,14.542,151.393
C08150=1103.878,188.925,-66.900,178.398,14.540,151.392
C08151=1103.884,189.174,-66.923,178.402,14.540,151.391
C08152=1103.889,189.422,-66.947,178.406,14.538,151.390
C08153=1103.895,189.671,-66.970,178.410,14.537,151.389
C08154=1103.900,189.920,-66.993,178.415,14.537,151.388
C08155=1103.906,190.169,-67.016,178.418,14.536,151.387
C08156=1103.912,190.417,-67.040,178.422,14.535,151.386
C08157=1103.917,190.666,-67.063,178.426,14.534,151.385
C08158=1103.923,190.915,-67.086,178.430,14.533,151.384
C08159=1103.928,191.164,-67.109,178.434,14.531,151.382
C08160=1103.934,191.413,-67.133,178.438,14.531,151.381
C08161=1103.940,191.662,-67.156,178.442,14.530,151.380
C08162=1103.946,191.934,-67.182,178.446,14.528,151.379
C08163=1103.952,192.205,-67.208,178.451,14.527,151.378
C08164=1103.959,192.476,-67.233,178.455,14.526,151.377
C08165=1103.964,192.748,-67.259,178.460,14.525,151.375
C08166=1103.970,192.997,-67.282,178.463,14.524,151.374
C08167=1103.976,193.246,-67.305,178.468,14.524,151.373
C08168=1103.981,193.494,-67.329,178.471,14.522,151.372
C08169=1103.987,193.743,-67.352,178.476,14.521,151.371
C08170=1103.993,193.992,-67.375,178.480,14.521,151.370
C08171=1103.998,194.241,-67.400,178.484,14.519,151.369
C08172=1104.005,194.490,-67.423,178.488,14.518,151.368
C08173=1104.011,194.738,-67.447,178.491,14.517,151.367
C08174=1104.016,194.988,-67.470,178.496,14.516,151.365
C08175=1104.022,195.236,-67.494,178.499,14.515,151.364
C08176=1104.027,195.485,-67.517,178.504,14.514,151.363
C08177=1104.033,195.733,-67.541,178.507,14.512,151.362
C08178=1104.039,195.983,-67.564,178.512,14.512,151.361
C08179=1104.044,196.232,-67.589,178.516,14.511,151.360
C08180=1104.050,196.481,-67.612,178.520,14.510,151.359
C08181=1104.055,196.729,-67.636,178.524,14.509,151.358
C08182=1104.061,196.977,-67.659,178.528,14.507,151.356
C08183=1104.068,197.227,-67.683,178.532,14.507,151.355
C08184=1104.073,197.476,-67.707,178.536,14.505,151.354
C08185=1104.079,197.724,-67.730,178.540,14.504,151.353
C08186=1104.084,197.973,-67.754,178.545,14.503,151.352
C08187=1104.090,198.221,-67.778,178.548,14.502,151.351
C08188=1104.096,198.471,-67.802,178.553,14.501,151.349
C08189=1104.102,198.719,-67.825,178.556,14.500,151.348
C08190=1104.107,198.968,-67.850,178.561,14.499,151.347
C08191=1104.113,199.217,-67.873,178.564,14.498,151.346
C08192=1104.119,199.466,-67.897,178.569,14.497,151.345
C08193=1104.125,199.715,-67.921,178.572,14.495,151.344
C08194=1104.130,199.964,-67.944,178.577,14.494,151.343
C08195=1104.136,200.213,-67.968,178.581,14.494,151.341
C08196=1104.142,200.461,-67.993,178.585,14.492,151.340
C08197=1104.148,200.710,-68.016,178.589,14.492,151.339
C08198=1104.153,200.958,-68.041,178.593,14.490,151.338
C08199=1104.159,201.208,-68.064,178.597,14.489,151.337
C08200=1104.165,201.456,-68.088,178.601,14.488,151.336
C08201=1104.171,201.705,-68.112,178.605,14.487,151.334
C08202=1104.176,201.954,-68.137,178.610,14.486,151.333
C08203=1104.183,202.202,-68.160,178.613,14.484,151.332
C08204=1104.187,202.451,-68.184,178.618,14.484,151.331
C08205=1104.194,202.700,-68.208,178.621,14.482,151.330
C08206=1104.199,202.949,-68.232,178.626,14.481,151.329
C08207=1104.205,203.198,-68.256,178.629,14.480,151.328
C08208=1104.211,203.447,-68.280,178.634,14.479,151.326
C08209=1104.217,203.695,-68.305,178.638,14.478,151.325
C08210=1104.222,203.944,-68.329,178.642,14.477,151.324
C08211=1104.228,204.192,-68.352,178.646,14.476,151.323
C08212=1104.234,204.442,-68.376,178.650,14.474,151.322
C08213=1104.239,204.691,-68.401,178.654,14.474,151.321
C08214=1104.244,204.939,-68.425,178.658,14.472,151.319
C08215=1104.251,205.188,-68.449,178.663,14.471,151.318
C08216=1104.256,205.437,-68.473,178.667,14.471,151.317
C08217=1104.261,205.685,-68.497,178.671,14.469,151.316
C08218=1104.267,205.935,-68.522,178.675,14.468,151.315
C08219=1104.273,206.183,-68.546,178.679,14.467,151.314
C08220=1104.279,206.432,-68.570,178.683,14.466,151.312
C08221=1104.285,206.681,-68.595,178.687,14.465,151.311
C08222=1104.290,206.929,-68.619,178.691,14.464,151.310
C08223=1104.297,207.178,-68.643,178.696,14.463,151.309
C08224=1104.302,207.426,-68.668,178.699,14.461,151.308
C08225=1104.307,207.675,-68.692,178.704,14.460,151.307
C08226=1104.330,208.673,-68.789,178.732,14.462,151.301
C08227=1104.338,209.041,-68.826,178.737,14.461,151.299
C08228=1104.347,209.407,-68.862,178.743,14.462,151.298
C08229=1104.356,209.774,-68.898,178.749,14.461,151.297
C08230=1104.364,210.142,-68.935,178.755,14.460,151.295
C08231=1104.370,210.390,-68.959,178.758,14.460,151.294
C08232=1104.376,210.640,-68.983,178.762,14.460,151.293
C08233=1104.381,210.888,-69.008,178.766,14.460,151.293
C08234=1104.387,211.136,-69.033,178.770,14.459,151.292
C08235=1104.392,211.386,-69.057,178.774,14.458,151.291
C08236=1104.398,211.634,-69.082,178.777,14.458,151.290
C08237=1104.404,211.883,-69.107,178.781,14.458,151.289
C08238=1104.409,212.131,-69.131,178.785,14.458,151.288
C08239=1104.415,212.381,-69.156,178.789,14.458,151.287
C08240=1104.421,212.629,-69.181,178.793,14.457,151.286
C08241=1104.427,212.878,-69.205,178.797,14.457,151.285
C08242=1104.432,213.126,-69.231,178.800,14.457,151.284
C08243=1104.437,213.376,-69.256,178.804,14.456,151.283
C08244=1104.443,213.624,-69.280,178.808,14.456,151.282
C08245=1104.449,213.873,-69.305,178.812,14.456,151.281
C08246=1104.454,214.121,-69.329,178.816,14.456,151.280
C08247=1104.460,214.370,-69.355,178.820,14.456,151.280
C08248=1104.466,214.619,-69.379,178.824,14.455,151.279
C08249=1104.472,214.868,-69.404,178.828,14.455,151.278
C08250=1104.477,215.116,-69.429,178.832,14.455,151.277
C08251=1104.482,215.365,-69.454,178.835,14.454,151.276
C08252=1104.488,215.613,-69.479,178.839,14.454,151.275
C08253=1104.494,215.863,-69.503,178.843,14.454,151.274
C08254=1104.500,216.111,-69.528,178.847,14.454,151.273
C08255=1104.505,216.360,-69.553,178.851,14.454,151.272
C08256=1104.511,216.609,-69.579,178.855,14.453,151.271
C08257=1104.516,216.857,-69.604,178.859,14.453,151.271
C08258=1104.522,217.106,-69.629,178.863,14.453,151.269
C08259=1104.528,217.354,-69.653,178.867,14.453,151.269
C08260=1104.533,217.604,-69.679,178.870,14.452,151.268
C08261=1104.539,217.852,-69.704,178.874,14.452,151.267
C08262=1104.545,218.100,-69.729,178.878,14.452,151.266
C08263=1104.551,218.350,-69.754,178.882,14.452,151.265
C08264=1104.556,218.598,-69.779,178.886,14.451,151.264
C08265=1104.562,218.847,-69.805,178.890,14.451,151.263
C08266=1104.567,219.095,-69.829,178.894,14.451,151.262
C08267=1104.573,219.344,-69.854,178.897,14.451,151.261
C08268=1104.579,219.593,-69.880,178.901,14.451,151.260
C08269=1104.584,219.841,-69.904,178.905,14.450,151.260
C08270=1104.590,220.090,-69.930,178.909,14.450,151.258
C08271=1104.597,220.339,-69.955,178.913,14.449,151.258
C08272=1104.601,220.588,-69.980,178.916,14.449,151.257
C08273=1104.607,220.836,-70.005,178.920,14.449,151.256
C08274=1104.614,221.085,-70.031,178.924,14.449,151.255
C08275=1104.618,221.333,-70.056,178.928,14.449,151.254
C08276=1104.625,221.582,-70.081,178.932,14.448,151.253
C08277=1104.631,221.831,-70.106,178.936,14.448,151.252
C08278=1104.635,222.080,-70.132,178.940,14.448,151.251
C08279=1104.644,222.450,-70.169,178.946,14.447,151.250
C08280=1104.653,222.821,-70.207,178.952,14.448,151.249
C08281=1104.660,223.192,-70.245,178.957,14.447,151.247
C08282=1104.670,223.562,-70.283,178.963,14.447,151.246
C08283=1104.675,223.810,-70.308,178.967,14.447,151.245
C08284=1104.680,224.059,-70.334,178.970,14.447,151.244
C08285=1104.687,224.308,-70.359,178.975,14.446,151.243
C08286=1104.692,224.557,-70.385,178.979,14.446,151.242
C08287=1104.698,224.805,-70.410,178.982,14.446,151.241
C08288=1104.703,225.054,-70.436,178.986,14.446,151.240
C08289=1104.709,225.303,-70.461,178.990,14.446,151.240
C08290=1104.714,225.551,-70.487,178.994,14.446,151.239
C08291=1104.720,225.800,-70.512,178.998,14.446,151.238
C08292=1104.726,226.048,-70.538,179.002,14.445,151.237
C08293=1104.732,226.297,-70.563,179.006,14.445,151.236
C08294=1104.737,226.545,-70.589,179.010,14.445,151.235
C08295=1104.743,226.794,-70.614,179.013,14.445,151.234
C08296=1104.749,227.043,-70.640,179.018,14.445,151.233
C08297=1104.754,227.292,-70.666,179.021,14.444,151.232
C08298=1104.760,227.540,-70.691,179.025,14.444,151.231
C08299=1104.765,227.788,-70.718,179.029,14.444,151.231
C08300=1104.772,228.037,-70.743,179.032,14.444,151.230
C08301=1104.777,228.286,-70.769,179.036,14.444,151.229
C08302=1104.783,228.535,-70.794,179.040,14.443,151.228
C08303=1104.788,228.783,-70.820,179.044,14.443,151.227
C08304=1104.794,229.032,-70.846,179.048,14.443,151.226
C08305=1104.800,229.281,-70.871,179.052,14.443,151.225
C08306=1104.806,229.529,-70.898,179.056,14.443,151.224
C08307=1104.811,229.778,-70.924,179.060,14.443,151.223
C08308=1104.817,230.027,-70.949,179.064,14.443,151.222
C08309=1104.822,230.275,-70.975,179.068,14.442,151.221
C08310=1104.829,230.523,-71.001,179.072,14.442,151.221
C08311=1104.834,230.772,-71.027,179.076,14.442,151.220
C08312=1104.840,231.021,-71.052,179.079,14.442,151.219
C08313=1104.845,231.270,-71.078,179.083,14.442,151.218
C08314=1104.852,231.518,-71.104,179.087,14.442,151.217
C08315=1104.856,231.766,-71.130,179.091,14.442,151.216
C08316=1104.862,232.015,-71.156,179.095,14.442,151.215
C08317=1104.867,232.264,-71.182,179.099,14.442,151.214
C08318=1104.874,232.512,-71.208,179.103,14.442,151.214
C08319=1104.879,232.761,-71.234,179.107,14.442,151.213
C08320=1104.885,233.010,-71.260,179.110,14.442,151.212
C08321=1104.891,233.259,-71.286,179.114,14.442,151.211
C08322=1104.895,233.507,-71.312,179.118,14.442,151.210
C08323=1104.902,233.755,-71.338,179.122,14.441,151.209
C08324=1104.907,234.004,-71.364,179.126,14.441,151.208
C08325=1104.913,234.253,-71.390,179.130,14.441,151.207
C08326=1104.919,234.501,-71.417,179.134,14.441,151.206
C08327=1104.924,234.750,-71.443,179.138,14.441,151.206
C08328=1104.930,234.999,-71.469,179.141,14.441,151.205
C08329=1104.935,235.248,-71.495,179.145,14.441,151.204
C08330=1104.942,235.496,-71.521,179.149,14.441,151.203
C08331=1104.950,235.858,-71.559,179.155,14.441,151.202
C08332=1104.958,236.220,-71.597,179.161,14.441,151.200
C08333=1104.966,236.583,-71.635,179.166,14.441,151.199
C08334=1104.974,236.944,-71.673,179.171,14.440,151.198
C08335=1104.980,237.192,-71.700,179.175,14.440,151.197
C08336=1104.985,237.441,-71.726,179.179,14.440,151.196
C08337=1104.991,237.690,-71.753,179.183,14.440,151.195
C08338=1104.997,237.939,-71.779,179.187,14.440,151.194
C08339=1105.002,238.187,-71.805,179.191,14.440,151.193
C08340=1105.008,238.435,-71.832,179.195,14.440,151.193
C08341=1105.014,238.684,-71.858,179.199,14.441,151.192
C08342=1105.019,238.933,-71.884,179.203,14.440,151.191
C08343=1105.025,239.181,-71.911,179.207,14.440,151.190
C08344=1105.031,239.430,-71.937,179.211,14.440,151.189
C08345=1105.036,239.678,-71.964,179.215,14.440,151.188
C08346=1105.042,239.927,-71.990,179.219,14.440,151.187
C08347=1105.048,240.176,-72.016,179.223,14.440,151.186
C08348=1105.053,240.424,-72.043,179.227,14.440,151.186
C08349=1105.059,240.672,-72.069,179.230,14.440,151.185
C08350=1105.065,240.921,-72.096,179.234,14.440,151.184
C08351=1105.070,241.170,-72.122,179.238,14.440,151.183
C08352=1105.076,241.418,-72.149,179.242,14.440,151.182
C08353=1105.082,241.666,-72.175,179.246,14.440,151.181
C08354=1105.088,241.915,-72.202,179.249,14.440,151.180
C08355=1105.093,242.164,-72.230,179.253,14.440,151.180
C08356=1105.099,242.413,-72.256,179.257,14.440,151.179
C08357=1105.105,242.662,-72.282,179.261,14.440,151.178
C08358=1105.110,242.910,-72.309,179.265,14.440,151.177
C08359=1105.116,243.158,-72.336,179.269,14.440,151.176
C08360=1105.122,243.407,-72.362,179.273,14.440,151.175
C08361=1105.128,243.655,-72.389,179.277,14.440,151.174
C08362=1105.134,243.903,-72.415,179.280,14.440,151.173
C08363=1105.139,244.152,-72.443,179.284,14.440,151.173
C08364=1105.144,244.400,-72.469,179.288,14.440,151.172
C08365=1105.150,244.649,-72.496,179.292,14.441,151.171
C08366=1105.156,244.898,-72.522,179.296,14.441,151.170
C08367=1105.161,245.146,-72.549,179.300,14.441,151.169
C08368=1105.167,245.395,-72.576,179.304,14.441,151.168
C08369=1105.173,245.644,-72.603,179.308,14.441,151.167
C08370=1105.179,245.892,-72.629,179.312,14.441,151.167
C08371=1105.184,246.141,-72.657,179.315,14.441,151.166
C08372=1105.189,246.389,-72.683,179.319,14.441,151.165
C08373=1105.195,246.637,-72.711,179.323,14.441,151.164
C08374=1105.201,246.885,-72.737,179.327,14.441,151.163
C08375=1105.206,247.134,-72.765,179.331,14.441,151.162
C08376=1105.212,247.382,-72.791,179.335,14.441,151.162
C08377=1105.218,247.631,-72.818,179.338,14.441,151.161
C08378=1105.223,247.880,-72.846,179.342,14.441,151.160
C08379=1105.229,248.128,-72.872,179.347,14.442,151.159
C08380=1105.234,248.377,-72.899,179.351,14.442,151.158
C08381=1105.240,248.625,-72.926,179.354,14.442,151.157
C08382=1105.245,248.874,-72.953,179.358,14.442,151.157
C08383=1105.254,249.229,-72.992,179.363,14.442,151.155
C08384=1105.262,249.584,-73.031,179.369,14.442,151.154
C08385=1105.269,249.940,-73.070,179.375,14.442,151.153
C08386=1105.278,250.296,-73.108,179.380,14.443,151.152
C08387=1105.283,250.544,-73.136,179.384,14.443,151.151
C08388=1105.289,250.792,-73.163,179.388,14.443,151.150
C08389=1105.295,251.041,-73.190,179.392,14.443,151.149
C08390=1105.300,251.290,-73.217,179.395,14.443,151.149
C08391=1105.306,251.538,-73.244,179.399,14.443,151.148
C08392=1105.311,251.786,-73.272,179.403,14.443,151.147
C08393=1105.317,252.034,-73.298,179.407,14.443,151.146
C08394=1105.323,252.284,-73.326,179.411,14.444,151.145
C08395=1105.329,252.532,-73.353,179.415,14.444,151.144
C08396=1105.334,252.780,-73.381,179.419,14.444,151.144
C08397=1105.339,253.029,-73.408,179.423,14.445,151.143
C08398=1105.345,253.277,-73.436,179.427,14.445,151.142
C08399=1105.350,253.526,-73.463,179.430,14.444,151.141
C08400=1105.357,253.774,-73.490,179.434,14.444,151.140
C08401=1105.362,254.022,-73.518,179.438,14.445,151.139
C08402=1105.368,254.271,-73.545,179.442,14.445,151.139
C08403=1105.373,254.520,-73.572,179.446,14.445,151.138
C08404=1105.379,254.768,-73.599,179.450,14.445,151.137
C08405=1105.384,255.016,-73.627,179.454,14.446,151.136
C08406=1105.390,255.265,-73.655,179.458,14.446,151.135
C08407=1105.396,255.513,-73.682,179.461,14.446,151.134
C08408=1105.401,255.762,-73.709,179.465,14.446,151.134
C08409=1105.408,256.010,-73.737,179.469,14.446,151.133
C08410=1105.413,256.258,-73.765,179.473,14.446,151.132
C08411=1105.418,256.507,-73.792,179.477,14.447,151.131
C08412=1105.425,256.755,-73.820,179.481,14.447,151.130
C08413=1105.430,257.004,-73.847,179.485,14.447,151.130
C08414=1105.436,257.252,-73.875,179.489,14.447,151.129
C08415=1105.442,257.501,-73.902,179.492,14.448,151.128
C08416=1105.447,257.749,-73.930,179.496,14.448,151.127
C08417=1105.453,257.997,-73.957,179.500,14.448,151.126
C08418=1105.459,258.246,-73.985,179.504,14.449,151.126
C08419=1105.464,258.494,-74.013,179.508,14.449,151.125
C08420=1105.470,258.742,-74.040,179.512,14.449,151.124
C08421=1105.476,258.991,-74.068,179.516,14.449,151.123
C08422=1105.481,259.240,-74.096,179.519,14.449,151.122
C08423=1105.488,259.488,-74.124,179.523,14.449,151.121
C08424=1105.493,259.736,-74.152,179.527,14.449,151.121
C08425=1105.498,259.985,-74.179,179.531,14.450,151.120
C08426=1105.504,260.233,-74.207,179.535,14.450,151.119
C08427=1105.510,260.481,-74.235,179.539,14.450,151.118
C08428=1105.516,260.730,-74.263,179.543,14.450,151.117
C08429=1105.522,260.978,-74.291,179.546,14.450,151.117
C08430=1105.527,261.226,-74.318,179.550,14.450,151.116
C08431=1105.533,261.475,-74.346,179.555,14.451,151.115
C08432=1105.539,261.723,-74.374,179.558,14.451,151.114
C08433=1105.545,261.972,-74.402,179.562,14.451,151.113
C08434=1105.551,262.220,-74.430,179.566,14.452,151.113
C08435=1105.559,262.573,-74.469,179.572,14.452,151.111
C08436=1105.567,262.925,-74.509,179.577,14.452,151.110
C08437=1105.575,263.278,-74.549,179.582,14.452,151.109
C08438=1105.583,263.631,-74.588,179.588,14.453,151.108
C08439=1105.589,263.880,-74.617,179.592,14.453,151.107
C08440=1105.594,264.128,-74.644,179.595,14.453,151.106
C08441=1105.601,264.376,-74.672,179.600,14.454,151.105
C08442=1105.606,264.624,-74.700,179.604,14.454,151.105
C08443=1105.612,264.873,-74.728,179.607,14.454,151.104
C08444=1105.618,265.121,-74.756,179.611,14.455,151.103
C08445=1105.624,265.370,-74.785,179.615,14.455,151.102
C08446=1105.629,265.618,-74.813,179.618,14.455,151.102
C08447=1105.635,265.866,-74.841,179.623,14.456,151.101
C08448=1105.640,266.114,-74.869,179.627,14.456,151.100
C08449=1105.646,266.363,-74.897,179.630,14.456,151.099
C08450=1105.651,266.611,-74.925,179.634,14.457,151.099
C08451=1105.658,266.859,-74.954,179.638,14.457,151.098
C08452=1105.663,267.107,-74.982,179.642,14.458,151.097
C08453=1105.669,267.356,-75.011,179.646,14.458,151.096
C08454=1105.674,267.604,-75.039,179.649,14.458,151.095
C08455=1105.680,267.853,-75.067,179.653,14.458,151.095
C08456=1105.686,268.101,-75.095,179.658,14.459,151.094
C08457=1105.692,268.350,-75.123,179.661,14.459,151.093
C08458=1105.697,268.597,-75.152,179.665,14.460,151.092
C08459=1105.702,268.846,-75.181,179.669,14.460,151.091
C08460=1105.708,269.094,-75.209,179.672,14.460,151.091
C08461=1105.714,269.343,-75.237,179.677,14.461,151.090
C08462=1105.719,269.591,-75.266,179.680,14.461,151.089
C08463=1105.725,269.839,-75.294,179.684,14.462,151.088
C08464=1105.731,270.088,-75.322,179.688,14.462,151.088
C08465=1105.737,270.336,-75.350,179.691,14.462,151.087
C08466=1105.743,270.584,-75.379,179.696,14.463,151.086
C08467=1105.748,270.832,-75.407,179.700,14.463,151.085
C08468=1105.753,271.081,-75.436,179.703,14.464,151.085
C08469=1105.759,271.329,-75.465,179.707,14.464,151.084
C08470=1105.765,271.578,-75.493,179.711,14.465,151.083
C08471=1105.771,271.826,-75.522,179.715,14.465,151.082
C08472=1105.777,272.074,-75.550,179.719,14.465,151.082
C08473=1105.782,272.323,-75.579,179.722,14.466,151.081
C08474=1105.787,272.570,-75.608,179.727,14.466,151.080
C08475=1105.793,272.819,-75.636,179.730,14.467,151.079
C08476=1105.799,273.068,-75.665,179.734,14.467,151.079
C08477=1105.805,273.315,-75.693,179.738,14.467,151.078
C08478=1105.810,273.564,-75.722,179.742,14.468,151.077
C08479=1105.816,273.812,-75.751,179.745,14.469,151.076
C08480=1105.822,274.060,-75.779,179.749,14.469,151.076
C08481=1105.828,274.309,-75.808,179.753,14.469,151.075
C08482=1105.833,274.557,-75.837,179.757,14.470,151.074
C08483=1105.839,274.805,-75.866,179.761,14.470,151.073
C08484=1105.845,275.054,-75.894,179.764,14.471,151.073
C08485=1105.850,275.301,-75.923,179.768,14.471,151.072
C08486=1105.856,275.550,-75.952,179.773,14.472,151.071
C08487=1105.864,275.906,-75.993,179.777,14.472,151.070
C08488=1105.872,276.261,-76.034,179.783,14.473,151.069
C08489=1105.880,276.617,-76.076,179.789,14.474,151.068
C08490=1105.888,276.972,-76.117,179.794,14.474,151.067
C08491=1105.894,277.220,-76.146,179.798,14.476,151.066
C08492=1105.900,277.469,-76.175,179.802,14.476,151.066
C08493=1105.905,277.717,-76.204,179.805,14.476,151.065
C08494=1105.911,277.965,-76.233,179.809,14.476,151.064
C08495=1105.917,278.213,-76.262,179.813,14.478,151.063
C08496=1105.923,278.462,-76.292,179.817,14.478,151.063
C08497=1105.928,278.710,-76.320,179.820,14.478,151.062
C08498=1105.933,278.958,-76.349,179.825,14.479,151.061
C08499=1105.940,279.206,-76.378,179.828,14.480,151.060
C08500=1105.945,279.454,-76.408,179.832,14.480,151.060
C08501=1105.951,279.703,-76.436,179.835,14.480,151.059
C08502=1105.956,279.951,-76.466,179.840,14.482,151.058
C08503=1105.962,280.199,-76.495,179.843,14.482,151.058
C08504=1105.967,280.447,-76.524,179.847,14.482,151.057
C08505=1105.973,280.695,-76.553,179.851,14.483,151.056
C08506=1105.979,280.944,-76.583,179.855,14.484,151.056
C08507=1105.985,281.192,-76.611,179.858,14.484,151.055
C08508=1105.990,281.441,-76.640,179.863,14.485,151.054
C08509=1105.996,281.688,-76.669,179.866,14.486,151.053
C08510=1106.002,281.937,-76.699,179.870,14.486,151.053
C08511=1106.008,282.185,-76.728,179.873,14.486,151.052
C08512=1106.013,282.433,-76.757,179.878,14.487,151.051
C08513=1106.018,282.681,-76.787,179.881,14.488,151.051
C08514=1106.025,282.929,-76.816,179.885,14.488,151.050
C08515=1106.030,283.178,-76.845,179.889,14.489,151.049
C08516=1106.036,283.426,-76.875,179.893,14.490,151.049
C08517=1106.041,283.673,-76.904,179.896,14.490,151.048
C08518=1106.047,283.922,-76.933,179.900,14.491,151.047
C08519=1106.052,284.170,-76.963,179.904,14.492,151.046
C08520=1106.058,284.418,-76.992,179.907,14.492,151.046
C08521=1106.064,284.667,-77.022,179.912,14.493,151.045
C08522=1106.069,284.915,-77.051,179.915,14.494,151.044
C08523=1106.075,285.163,-77.080,179.919,14.494,151.044
C08524=1106.081,285.411,-77.110,179.923,14.495,151.043
C08525=1106.086,285.660,-77.139,179.926,14.496,151.042
C08526=1106.092,285.908,-77.168,179.930,14.496,151.042
C08527=1106.098,286.156,-77.199,179.934,14.497,151.041
C08528=1106.104,286.404,-77.228,179.938,14.498,151.040
C08529=1106.109,286.653,-77.258,179.941,14.498,151.040
C08530=1106.115,286.900,-77.287,179.946,14.499,151.039
C08531=1106.120,287.148,-77.316,179.949,14.500,151.038
C08532=1106.126,287.396,-77.347,179.953,14.501,151.038
C08533=1106.132,287.645,-77.376,179.957,14.501,151.037
C08534=1106.138,287.893,-77.405,179.960,14.502,151.036
C08535=1106.143,288.141,-77.435,179.965,14.503,151.036
C08536=1106.149,288.389,-77.465,179.968,14.503,151.035
C08537=1106.155,288.638,-77.495,179.972,14.504,151.034
C08538=1106.161,288.886,-77.524,179.976,14.505,151.034
C08539=1106.169,289.250,-77.567,179.981,14.506,151.033
C08540=1106.178,289.615,-77.611,179.987,14.507,151.032
C08541=1106.186,289.980,-77.655,179.992,14.508,151.031
C08542=1106.194,290.345,-77.700,179.997,14.509,151.030
C08543=1106.200,290.594,-77.729,-179.999,14.510,151.029
C08544=1106.206,290.842,-77.758,-179.995,14.511,151.028
C08545=1106.212,291.090,-77.789,-179.991,14.512,151.028
C08546=1106.217,291.338,-77.818,-179.987,14.512,151.027
C08547=1106.223,291.586,-77.849,-179.984,14.513,151.026
C08548=1106.228,291.834,-77.878,-179.980,14.514,151.026
C08549=1106.234,292.082,-77.909,-179.976,14.515,151.025
C08550=1106.240,292.331,-77.938,-179.972,14.516,151.025
C08551=1106.245,292.578,-77.968,-179.969,14.516,151.024
C08552=1106.250,292.826,-77.998,-179.965,14.517,151.023
C08553=1106.256,293.074,-78.028,-179.961,14.518,151.023
C08554=1106.262,293.322,-78.058,-179.958,14.519,151.022
C08555=1106.268,293.570,-78.088,-179.953,14.520,151.021
C08556=1106.273,293.819,-78.118,-179.950,14.520,151.021
C08557=1106.279,294.066,-78.148,-179.947,14.521,151.020
C08558=1106.284,294.315,-78.178,-179.943,14.522,151.019
C08559=1106.290,294.563,-78.208,-179.939,14.523,151.019
C08560=1106.296,294.811,-78.239,-179.935,14.524,151.018
C08561=1106.302,295.059,-78.268,-179.932,14.525,151.018
C08562=1106.307,295.307,-78.299,-179.928,14.525,151.017
C08563=1106.313,295.555,-78.328,-179.924,14.527,151.016
C08564=1106.319,295.804,-78.359,-179.921,14.527,151.016
C08565=1106.325,296.052,-78.389,-179.916,14.529,151.015
C08566=1106.331,296.299,-78.420,-179.913,14.529,151.014
C08567=1106.337,296.548,-78.449,-179.909,14.531,151.014
C08568=1106.342,296.796,-78.480,-179.905,14.531,151.013
C08569=1106.347,297.044,-78.510,-179.902,14.531,151.013
C08570=1106.353,297.292,-78.540,-179.898,14.533,151.012
C08571=1106.359,297.540,-78.570,-179.895,14.533,151.011
C08572=1106.365,297.788,-78.601,-179.891,14.535,151.011
C08573=1106.370,298.036,-78.631,-179.887,14.535,151.010
C08574=1106.376,298.284,-78.662,-179.883,14.537,151.010
C08575=1106.381,298.532,-78.692,-179.880,14.538,151.009
C08576=1106.387,298.780,-78.722,-179.875,14.539,151.008
C08577=1106.393,299.028,-78.752,-179.872,14.540,151.008
C08578=1106.398,299.276,-78.783,-179.868,14.541,151.007
C08579=1106.404,299.524,-78.814,-179.865,14.542,151.007
C08580=1106.409,299.772,-78.844,-179.861,14.543,151.006
C08581=1106.414,300.020,-78.875,-179.857,14.544,151.006
C08582=1106.420,300.268,-78.905,-179.853,14.545,151.005
C08583=1106.426,300.516,-78.935,-179.850,14.546,151.004
C08584=1106.431,300.765,-78.966,-179.847,14.546,151.004
C08585=1106.437,301.013,-78.997,-179.843,14.548,151.003
C08586=1106.443,301.261,-79.027,-179.839,14.548,151.003
C08587=1106.448,301.509,-79.058,-179.835,14.550,151.002
C08588=1106.454,301.757,-79.088,-179.832,14.551,151.002
C08589=1106.460,302.004,-79.119,-179.828,14.552,151.001
C08590=1106.465,302.252,-79.150,-179.825,14.553,151.001
C08591=1106.474,302.631,-79.197,-179.818,14.555,151.000
C08592=1106.482,303.010,-79.243,-179.813,14.556,150.999
C08593=1106.491,303.389,-79.290,-179.807,14.558,150.998
C08594=1106.500,303.768,-79.337,-179.802,14.560,150.997
C08595=1106.505,304.016,-79.368,-179.799,14.561,150.997
C08596=1106.511,304.264,-79.399,-179.794,14.562,150.996
C08597=1106.516,304.512,-79.430,-179.791,14.563,150.995
C08598=1106.522,304.760,-79.460,-179.787,14.564,150.995
C08599=1106.528,305.008,-79.492,-179.784,14.565,150.994
C08600=1106.533,305.256,-79.522,-179.780,14.566,150.994
C08601=1106.538,305.504,-79.553,-179.776,14.568,150.993
C08602=1106.545,305.752,-79.584,-179.773,14.569,150.993
C08603=1106.551,306.000,-79.614,-179.769,14.570,150.992
C08604=1106.556,306.248,-79.646,-179.765,14.571,150.992
C08605=1106.562,306.495,-79.676,-179.762,14.572,150.991
C08606=1106.568,306.744,-79.707,-179.758,14.573,150.990
C08607=1106.573,306.992,-79.738,-179.754,14.574,150.990
C08608=1106.579,307.240,-79.769,-179.751,14.575,150.989
C08609=1106.585,307.487,-79.800,-179.747,14.577,150.989
C08610=1106.590,307.736,-79.831,-179.744,14.578,150.988
C08611=1106.596,307.984,-79.863,-179.740,14.579,150.988
C08612=1106.601,308.232,-79.893,-179.736,14.580,150.987
C08613=1106.607,308.480,-79.924,-179.733,14.581,150.987
C08614=1106.613,308.728,-79.955,-179.729,14.583,150.986
C08615=1106.618,308.976,-79.986,-179.725,14.583,150.986
C08616=1106.624,309.223,-80.017,-179.721,14.585,150.985
C08617=1106.630,309.472,-80.049,-179.718,14.586,150.985
C08618=1106.636,309.720,-80.079,-179.714,14.587,150.984
C08619=1106.641,309.967,-80.111,-179.711,14.588,150.984
C08620=1106.647,310.216,-80.142,-179.707,14.590,150.983
C08621=1106.653,310.463,-80.173,-179.704,14.590,150.982
C08622=1106.658,310.711,-80.204,-179.700,14.592,150.982
C08623=1106.665,310.959,-80.235,-179.696,14.593,150.981
C08624=1106.670,311.207,-80.266,-179.693,14.594,150.981
C08625=1106.675,311.455,-80.298,-179.689,14.596,150.981
C08626=1106.682,311.703,-80.329,-179.686,14.597,150.980
C08627=1106.687,311.951,-80.360,-179.682,14.598,150.980
C08628=1106.693,312.199,-80.392,-179.678,14.599,150.979
C08629=1106.699,312.447,-80.423,-179.675,14.601,150.979
C08630=1106.704,312.694,-80.454,-179.671,14.602,150.978
C08631=1106.710,312.943,-80.486,-179.667,14.603,150.977
C08632=1106.716,313.190,-80.517,-179.663,14.604,150.977
C08633=1106.722,313.439,-80.549,-179.660,14.605,150.976
C08634=1106.727,313.687,-80.580,-179.656,14.607,150.976
C08635=1106.733,313.934,-80.611,-179.653,14.608,150.975
C08636=1106.739,314.182,-80.643,-179.649,14.609,150.975
C08637=1106.744,314.430,-80.674,-179.646,14.610,150.974
C08638=1106.751,314.678,-80.705,-179.642,14.612,150.974
C08639=1106.757,314.926,-80.737,-179.638,14.613,150.973
C08640=1106.762,315.175,-80.768,-179.635,14.614,150.973
C08641=1106.768,315.422,-80.800,-179.631,14.616,150.972
C08642=1106.774,315.670,-80.832,-179.628,14.617,150.972
C08643=1106.782,316.051,-80.880,-179.622,14.619,150.971
C08644=1106.791,316.433,-80.929,-179.616,14.622,150.971
C08645=1106.799,316.814,-80.977,-179.612,14.624,150.970
C08646=1106.808,317.196,-81.026,-179.606,14.626,150.969
C08647=1106.813,317.444,-81.058,-179.603,14.627,150.969
C08648=1106.819,317.691,-81.090,-179.599,14.629,150.968
C08649=1106.825,317.940,-81.122,-179.595,14.631,150.968
C08650=1106.830,318.187,-81.153,-179.592,14.632,150.968
C08651=1106.836,318.436,-81.185,-179.588,14.633,150.967
C08652=1106.841,318.683,-81.216,-179.585,14.635,150.967
C08653=1106.847,318.932,-81.248,-179.581,14.636,150.966
C08654=1106.853,319.179,-81.280,-179.578,14.638,150.966
C08655=1106.859,319.427,-81.312,-179.574,14.640,150.966
C08656=1106.864,319.675,-81.344,-179.571,14.641,150.965
C08657=1106.870,319.923,-81.376,-179.567,14.642,150.965
C08658=1106.875,320.171,-81.407,-179.563,14.644,150.964
C08659=1106.881,320.419,-81.440,-179.560,14.645,150.964
C08660=1106.886,320.667,-81.472,-179.557,14.647,150.963
C08661=1106.892,320.915,-81.504,-179.553,14.649,150.963
C08662=1106.897,321.162,-81.535,-179.550,14.650,150.963
C08663=1106.903,321.411,-81.567,-179.546,14.651,150.962
C08664=1106.909,321.658,-81.599,-179.542,14.653,150.962
C08665=1106.915,321.906,-81.631,-179.539,14.654,150.961
C08666=1106.920,322.154,-81.663,-179.536,14.656,150.961
C08667=1106.926,322.402,-81.695,-179.532,14.658,150.961
C08668=1106.932,322.650,-81.728,-179.529,14.659,150.960
C08669=1106.937,322.897,-81.760,-179.525,14.661,150.960
C08670=1106.943,323.146,-81.792,-179.521,14.663,150.959
C08671=1106.948,323.393,-81.823,-179.518,14.664,150.959
C08672=1106.954,323.641,-81.855,-179.515,14.666,150.959
C08673=1106.960,323.889,-81.887,-179.511,14.667,150.958
C08674=1106.965,324.137,-81.920,-179.508,14.668,150.958
C08675=1106.971,324.385,-81.952,-179.504,14.670,150.958
C08676=1106.977,324.633,-81.984,-179.501,14.672,150.957
C08677=1106.983,324.881,-82.016,-179.498,14.673,150.957
C08678=1106.989,325.129,-82.048,-179.494,14.675,150.956
C08679=1106.994,325.376,-82.081,-179.490,14.677,150.956
C08680=1107.000,325.624,-82.113,-179.487,14.679,150.956
C08681=1107.006,325.873,-82.145,-179.483,14.680,150.955
C08682=1107.011,326.119,-82.177,-179.480,14.682,150.955
C08683=1107.017,326.368,-82.210,-179.476,14.683,150.954
C08684=1107.022,326.616,-82.242,-179.472,14.685,150.954
C08685=1107.028,326.863,-82.275,-179.470,14.687,150.954
C08686=1107.034,327.111,-82.307,-179.466,14.688,150.953
C08687=1107.039,327.360,-82.339,-179.462,14.690,150.953
C08688=1107.045,327.607,-82.372,-179.459,14.691,150.953
C08689=1107.051,327.855,-82.404,-179.456,14.693,150.952
C08690=1107.057,328.103,-82.437,-179.452,14.695,150.952
C08691=1107.063,328.351,-82.469,-179.448,14.697,150.952
C08692=1107.068,328.598,-82.501,-179.445,14.698,150.951
C08693=1107.074,328.846,-82.533,-179.442,14.700,150.951
C08694=1107.080,329.094,-82.567,-179.438,14.702,150.950
C08695=1107.088,329.469,-82.615,-179.433,14.705,150.950
C08696=1107.097,329.843,-82.664,-179.428,14.707,150.949
C08697=1107.106,330.218,-82.714,-179.422,14.710,150.949
C08698=1107.115,330.592,-82.763,-179.417,14.713,150.948
C08699=1107.120,330.839,-82.795,-179.414,14.714,150.948
C08700=1107.126,331.088,-82.828,-179.411,14.716,150.948
C08701=1107.132,331.335,-82.861,-179.407,14.718,150.947
C08702=1107.138,331.583,-82.893,-179.403,14.720,150.947
C08703=1107.143,331.831,-82.926,-179.400,14.721,150.947
C08704=1107.150,332.079,-82.959,-179.397,14.723,150.946
C08705=1107.155,332.326,-82.992,-179.393,14.725,150.946
C08706=1107.161,332.574,-83.024,-179.390,14.727,150.946
C08707=1107.166,332.822,-83.057,-179.386,14.729,150.945
C08708=1107.172,333.070,-83.090,-179.383,14.731,150.945
C08709=1107.177,333.318,-83.122,-179.380,14.732,150.945
C08710=1107.183,333.565,-83.155,-179.376,14.734,150.945
C08711=1107.189,333.813,-83.188,-179.373,14.736,150.944
C08712=1107.194,334.062,-83.221,-179.369,14.738,150.944
C08713=1107.201,334.309,-83.253,-179.366,14.740,150.944
C08714=1107.205,334.556,-83.286,-179.363,14.742,150.943
C08715=1107.212,334.804,-83.319,-179.359,14.744,150.943
C08716=1107.217,335.052,-83.352,-179.356,14.746,150.943
C08717=1107.223,335.300,-83.385,-179.353,14.748,150.943
C08718=1107.229,335.548,-83.418,-179.349,14.750,150.942
C08719=1107.234,335.796,-83.451,-179.346,14.752,150.942
C08720=1107.239,336.043,-83.484,-179.342,14.754,150.942
C08721=1107.246,336.291,-83.517,-179.339,14.756,150.942
C08722=1107.251,336.539,-83.550,-179.336,14.758,150.941
C08723=1107.257,336.787,-83.584,-179.332,14.760,150.941
C08724=1107.263,337.034,-83.616,-179.329,14.762,150.941
C08725=1107.269,337.282,-83.650,-179.326,14.764,150.941
C08726=1107.274,337.531,-83.682,-179.322,14.766,150.940
C08727=1107.280,337.778,-83.715,-179.318,14.768,150.940
C08728=1107.285,338.025,-83.748,-179.315,14.770,150.940
C08729=1107.291,338.273,-83.781,-179.312,14.772,150.940
C08730=1107.296,338.521,-83.815,-179.309,14.774,150.939
C08731=1107.303,338.769,-83.847,-179.306,14.776,150.939
C08732=1107.308,339.017,-83.881,-179.302,14.778,150.939
C08733=1107.314,339.264,-83.915,-179.299,14.780,150.939
C08734=1107.319,339.512,-83.948,-179.295,14.782,150.938
C08735=1107.325,339.760,-83.981,-179.292,14.785,150.938
C08736=1107.331,340.007,-84.014,-179.288,14.787,150.938
C08737=1107.337,340.255,-84.048,-179.285,14.789,150.938
C08738=1107.342,340.502,-84.081,-179.282,14.791,150.938
C08739=1107.347,340.750,-84.114,-179.279,14.793,150.937
C08740=1107.353,340.998,-84.147,-179.276,14.795,150.937
C08741=1107.358,341.246,-84.181,-179.272,14.797,150.937
C08742=1107.364,341.493,-84.215,-179.269,14.799,150.937
C08743=1107.371,341.741,-84.247,-179.266,14.802,150.937
C08744=1107.376,341.989,-84.281,-179.262,14.804,150.936
C08745=1107.382,342.237,-84.314,-179.259,14.806,150.936
C08746=1107.387,342.485,-84.347,-179.256,14.808,150.936
C08747=1107.396,342.852,-84.398,-179.251,14.812,150.936
C08748=1107.405,343.221,-84.447,-179.246,14.815,150.935
C08749=1107.413,343.589,-84.497,-179.241,14.819,150.935
C08750=1107.421,343.958,-84.547,-179.236,14.822,150.935
C08751=1107.427,344.206,-84.581,-179.232,14.824,150.935
C08752=1107.433,344.453,-84.615,-179.230,14.826,150.935
C08753=1107.438,344.701,-84.648,-179.226,14.828,150.934
C08754=1107.444,344.948,-84.682,-179.223,14.830,150.934
C08755=1107.450,345.196,-84.715,-179.220,14.833,150.934
C08756=1107.455,345.444,-84.749,-179.217,14.835,150.934
C08757=1107.461,345.691,-84.783,-179.213,14.838,150.934
C08758=1107.466,345.939,-84.816,-179.210,14.840,150.934
C08759=1107.472,346.187,-84.850,-179.207,14.842,150.934
C08760=1107.478,346.434,-84.883,-179.204,14.845,150.933
C08761=1107.484,346.682,-84.917,-179.200,14.847,150.933
C08762=1107.489,346.930,-84.951,-179.197,14.849,150.933
C08763=1107.495,347.177,-84.985,-179.194,14.852,150.933
C08764=1107.501,347.425,-85.018,-179.191,14.854,150.933
C08765=1107.507,347.672,-85.052,-179.187,14.857,150.933
C08766=1107.511,347.920,-85.086,-179.184,14.860,150.933
C08767=1107.517,348.168,-85.120,-179.180,14.862,150.933
C08768=1107.523,348.415,-85.154,-179.177,14.864,150.932
C08769=1107.529,348.663,-85.188,-179.174,14.867,150.932
C08770=1107.535,348.911,-85.221,-179.171,14.869,150.932
C08771=1107.541,349.159,-85.255,-179.168,14.872,150.932
C08772=1107.546,349.406,-85.290,-179.164,14.874,150.932
C08773=1107.551,349.654,-85.323,-179.161,14.877,150.932
C08774=1107.557,349.901,-85.357,-179.158,14.879,150.932
C08775=1107.563,350.149,-85.391,-179.155,14.882,150.932
C08776=1107.569,350.397,-85.425,-179.152,14.884,150.932
C08777=1107.574,350.644,-85.459,-179.148,14.886,150.931
C08778=1107.580,350.892,-85.494,-179.146,14.889,150.932
C08779=1107.585,351.139,-85.528,-179.142,14.891,150.931
C08780=1107.592,351.387,-85.561,-179.139,14.894,150.931
C08781=1107.597,351.635,-85.596,-179.136,14.897,150.931
C08782=1107.603,351.882,-85.630,-179.133,14.899,150.931
C08783=1107.608,352.130,-85.664,-179.129,14.902,150.931
C08784=1107.614,352.377,-85.699,-179.126,14.905,150.931
C08785=1107.619,352.625,-85.732,-179.123,14.907,150.931
C08786=1107.625,352.872,-85.766,-179.120,14.910,150.931
C08787=1107.631,353.120,-85.800,-179.117,14.912,150.931
C08788=1107.637,353.368,-85.835,-179.114,14.915,150.931
C08789=1107.642,353.615,-85.869,-179.111,14.918,150.931
C08790=1107.648,353.862,-85.903,-179.107,14.920,150.931
C08791=1107.653,354.110,-85.938,-179.105,14.923,150.931
C08792=1107.659,354.357,-85.972,-179.101,14.925,150.931
C08793=1107.665,354.606,-86.006,-179.098,14.929,150.931
C08794=1107.671,354.854,-86.040,-179.095,14.931,150.931
C08795=1107.676,355.101,-86.074,-179.092,14.934,150.931
C08796=1107.682,355.348,-86.109,-179.089,14.936,150.931
C08797=1107.687,355.596,-86.143,-179.085,14.939,150.931
C08798=1107.693,355.844,-86.178,-179.083,14.942,150.931
C08799=1107.702,356.214,-86.229,-179.077,14.946,150.931
C08800=1107.710,356.585,-86.281,-179.073,14.950,150.931
C08801=1107.718,356.954,-86.333,-179.068,14.954,150.931
C08802=1107.727,357.325,-86.384,-179.064,14.958,150.931
C08803=1107.732,357.572,-86.419,-179.061,14.961,150.931
C08804=1107.739,357.820,-86.453,-179.057,14.964,150.931
C08805=1107.744,358.068,-86.488,-179.054,14.967,150.931
C08806=1107.750,358.315,-86.522,-179.052,14.970,150.931
C08807=1107.755,358.563,-86.557,-179.048,14.972,150.931
C08808=1107.762,358.810,-86.592,-179.045,14.975,150.931
C08809=1107.767,359.058,-86.627,-179.042,14.978,150.931
C08810=1107.773,359.305,-86.661,-179.039,14.981,150.931
C08811=1107.778,359.553,-86.695,-179.036,14.984,150.931
C08812=1107.784,359.800,-86.731,-179.033,14.987,150.931
C08813=1107.790,360.048,-86.765,-179.030,14.990,150.931
C08814=1107.795,360.295,-86.800,-179.027,14.992,150.931
C08815=1107.801,360.543,-86.834,-179.024,14.996,150.931
C08816=1107.807,360.790,-86.869,-179.021,14.999,150.931
C08817=1107.812,361.038,-86.904,-179.018,15.001,150.931
C08818=1107.818,361.285,-86.938,-179.015,15.004,150.931
C08819=1107.824,361.533,-86.974,-179.011,15.008,150.931
C08820=1107.829,361.780,-87.009,-179.009,15.011,150.931
C08821=1107.835,362.028,-87.043,-179.006,15.014,150.932
C08822=1107.841,362.275,-87.078,-179.003,15.016,150.932
C08823=1107.846,362.523,-87.113,-178.999,15.020,150.932
C08824=1107.852,362.769,-87.148,-178.997,15.023,150.932
C08825=1107.858,363.018,-87.183,-178.994,15.026,150.932
C08826=1107.863,363.265,-87.218,-178.991,15.028,150.932
C08827=1107.868,363.512,-87.253,-178.987,15.032,150.932
C08828=1107.875,363.760,-87.288,-178.985,15.035,150.932
C08829=1107.880,364.007,-87.323,-178.982,15.038,150.932
C08830=1107.886,364.254,-87.358,-178.979,15.041,150.932
C08831=1107.891,364.503,-87.393,-178.976,15.044,150.933
C08832=1107.898,364.749,-87.428,-178.973,15.047,150.933
C08833=1107.903,364.997,-87.462,-178.970,15.050,150.933
C08834=1107.909,365.244,-87.498,-178.967,15.054,150.933
C08835=1107.914,365.492,-87.533,-178.964,15.057,150.933
C08836=1107.920,365.740,-87.568,-178.961,15.060,150.933
C08837=1107.926,365.986,-87.603,-178.959,15.063,150.933
C08838=1107.931,366.234,-87.638,-178.955,15.066,150.933
C08839=1107.937,366.482,-87.674,-178.952,15.069,150.934
C08840=1107.943,366.729,-87.709,-178.950,15.073,150.934
C08841=1107.948,366.977,-87.744,-178.946,15.076,150.934
C08842=1107.954,367.224,-87.779,-178.944,15.079,150.934
C08843=1107.959,367.471,-87.815,-178.941,15.082,150.934
C08844=1107.965,367.719,-87.850,-178.937,15.086,150.934
C08845=1107.970,367.966,-87.885,-178.935,15.089,150.935
C08846=1107.976,368.213,-87.920,-178.932,15.092,150.935
C08847=1107.982,368.461,-87.956,-178.929,15.096,150.935
C08848=1107.987,368.708,-87.991,-178.926,15.099,150.935
C08849=1107.993,368.956,-88.027,-178.923,15.103,150.936
C08850=1107.998,369.203,-88.062,-178.920,15.106,150.936
C08851=1108.008,369.588,-88.117,-178.916,15.111,150.936
C08852=1108.016,369.973,-88.172,-178.912,15.116,150.936
C08853=1108.026,370.358,-88.227,-178.907,15.121,150.937
C08854=1108.034,370.744,-88.282,-178.902,15.127,150.937
C08855=1108.040,370.991,-88.318,-178.900,15.130,150.937
C08856=1108.046,371.238,-88.353,-178.897,15.134,150.937
C08857=1108.051,371.485,-88.389,-178.894,15.137,150.938
C08858=1108.057,371.733,-88.425,-178.891,15.141,150.938
C08859=1108.063,371.980,-88.460,-178.888,15.144,150.938
C08860=1108.069,372.228,-88.496,-178.886,15.147,150.939
C08861=1108.073,372.475,-88.532,-178.883,15.151,150.939
C08862=1108.080,372.723,-88.567,-178.880,15.154,150.939
C08863=1108.085,372.970,-88.603,-178.877,15.158,150.939
C08864=1108.091,373.217,-88.638,-178.874,15.162,150.940
C08865=1108.096,373.464,-88.674,-178.871,15.166,150.940
C08866=1108.102,373.712,-88.710,-178.869,15.169,150.940
C08867=1108.108,373.959,-88.745,-178.866,15.172,150.940
C08868=1108.114,374.207,-88.781,-178.863,15.176,150.941
C08869=1108.120,374.453,-88.817,-178.860,15.179,150.941
C08870=1108.125,374.701,-88.853,-178.857,15.183,150.941
C08871=1108.130,374.948,-88.888,-178.855,15.187,150.942
C08872=1108.136,375.196,-88.924,-178.852,15.191,150.942
C08873=1108.142,375.443,-88.959,-178.849,15.194,150.942
C08874=1108.147,375.691,-88.996,-178.846,15.198,150.943
C08875=1108.153,375.937,-89.032,-178.844,15.202,150.943
C08876=1108.159,376.185,-89.068,-178.841,15.206,150.943
C08877=1108.164,376.432,-89.103,-178.838,15.209,150.944
C08878=1108.170,376.680,-89.139,-178.836,15.213,150.944
C08879=1108.176,376.927,-89.176,-178.833,15.216,150.944
C08880=1108.181,377.174,-89.211,-178.830,15.221,150.945
C08881=1108.187,377.422,-89.247,-178.828,15.224,150.945
C08882=1108.192,377.668,-89.284,-178.825,15.228,150.945
C08883=1108.198,377.916,-89.319,-178.822,15.232,150.946
C08884=1108.203,378.163,-89.355,-178.819,15.236,150.946
C08885=1108.209,378.410,-89.392,-178.817,15.239,150.946
C08886=1108.215,378.658,-89.427,-178.814,15.243,150.947
C08887=1108.220,378.905,-89.463,-178.812,15.247,150.947
C08888=1108.226,379.152,-89.500,-178.809,15.251,150.948
C08889=1108.232,379.399,-89.535,-178.806,15.255,150.948
C08890=1108.238,379.646,-89.572,-178.803,15.259,150.948
C08891=1108.244,379.894,-89.608,-178.800,15.263,150.949
C08892=1108.249,380.140,-89.644,-178.798,15.267,150.949
C08893=1108.255,380.388,-89.680,-178.795,15.271,150.950
C08894=1108.261,380.635,-89.717,-178.793,15.274,150.950
C08895=1108.266,380.883,-89.753,-178.790,15.279,150.950
C08896=1108.272,381.130,-89.789,-178.788,15.282,150.951
C08897=1108.277,381.377,-89.825,-178.785,15.286,150.951
C08898=1108.283,381.624,-89.862,-178.782,15.291,150.952
C08899=1108.289,381.871,-89.898,-178.780,15.294,150.952
C08900=1108.294,382.118,-89.934,-178.777,15.299,150.953
C08901=1108.300,382.365,-89.970,-178.774,15.302,150.953
C08902=1108.306,382.613,-90.007,-178.771,15.306,150.953
C08903=1108.315,383.025,-90.067,-178.767,15.313,150.954
C08904=1108.325,383.437,-90.128,-178.763,15.320,150.955
C08905=1108.334,383.848,-90.189,-178.759,15.327,150.956
C08906=1108.344,384.260,-90.249,-178.754,15.334,150.957
C08907=1108.349,384.507,-90.286,-178.752,15.339,150.957
C08908=1108.354,384.755,-90.322,-178.749,15.342,150.958
C08909=1108.361,385.002,-90.359,-178.747,15.347,150.958
C08910=1108.366,385.249,-90.396,-178.744,15.352,150.959
C08911=1108.371,385.496,-90.433,-178.742,15.355,150.959
C08912=1108.377,385.743,-90.469,-178.739,15.360,150.960
C08913=1108.383,385.991,-90.505,-178.736,15.364,150.960
C08914=1108.388,386.238,-90.542,-178.735,15.368,150.961
C08915=1108.394,386.485,-90.578,-178.732,15.373,150.961
C08916=1108.400,386.732,-90.615,-178.729,15.377,150.962
C08917=1108.405,386.979,-90.652,-178.727,15.381,150.962
C08918=1108.411,387.226,-90.689,-178.724,15.385,150.963
C08919=1108.417,387.473,-90.726,-178.722,15.390,150.963
C08920=1108.422,387.720,-90.763,-178.719,15.395,150.964
C08921=1108.428,387.967,-90.799,-178.717,15.398,150.965
C08922=1108.434,388.214,-90.836,-178.714,15.403,150.965
C08923=1108.439,388.462,-90.873,-178.712,15.408,150.966
C08924=1108.445,388.709,-90.910,-178.709,15.412,150.966
C08925=1108.450,388.955,-90.946,-178.707,15.416,150.967
C08926=1108.456,389.203,-90.983,-178.705,15.421,150.968
C08927=1108.462,389.450,-91.020,-178.702,15.426,150.968
C08928=1108.467,389.697,-91.057,-178.699,15.430,150.969
C08929=1108.474,389.944,-91.093,-178.697,15.434,150.969
C08930=1108.479,390.192,-91.131,-178.695,15.439,150.970
C08931=1108.484,390.438,-91.167,-178.692,15.444,150.971
C08932=1108.490,390.686,-91.204,-178.689,15.448,150.971
C08933=1108.495,390.933,-91.241,-178.687,15.453,150.972
C08934=1108.502,391.180,-91.278,-178.685,15.457,150.972
C08935=1108.508,391.427,-91.315,-178.682,15.462,150.973
C08936=1108.513,391.674,-91.353,-178.680,15.467,150.974
C08937=1108.519,391.922,-91.390,-178.677,15.471,150.974
C08938=1108.524,392.168,-91.426,-178.675,15.476,150.975
C08939=1108.530,392.415,-91.463,-178.673,15.480,150.976
C08940=1108.536,392.662,-91.500,-178.671,15.485,150.976
C08941=1108.542,392.910,-91.537,-178.668,15.490,150.977
C08942=1108.547,393.157,-91.575,-178.666,15.495,150.978
C08943=1108.553,393.404,-91.612,-178.663,15.499,150.978
C08944=1108.559,393.651,-91.649,-178.662,15.504,150.979
C08945=1108.564,393.898,-91.686,-178.659,15.509,150.980
C08946=1108.570,394.146,-91.723,-178.657,15.514,150.981
C08947=1108.575,394.392,-91.761,-178.655,15.518,150.981
C08948=1108.581,394.639,-91.798,-178.652,15.523,150.982
C08949=1108.586,394.886,-91.835,-178.650,15.528,150.983
C08950=1108.592,395.133,-91.873,-178.647,15.533,150.984
C08951=1108.598,395.381,-91.910,-178.645,15.538,150.984
C08952=1108.604,395.628,-91.947,-178.643,15.543,150.985
C08953=1108.609,395.875,-91.984,-178.641,15.548,150.986
C08954=1108.614,396.122,-92.022,-178.639,15.552,150.986
C08955=1108.620,396.334,-92.054,-178.637,15.557,150.987
C08956=1108.625,396.546,-92.086,-178.635,15.562,150.988
C08957=1108.629,396.757,-92.118,-178.633,15.566,150.988
C08958=1108.634,396.970,-92.150,-178.631,15.570,150.989
C08959=1108.639,397.181,-92.183,-178.629,15.574,150.990
C08960=1108.644,397.394,-92.214,-178.627,15.579,150.991
C08961=1108.648,397.605,-92.247,-178.625,15.583,150.991
C08962=1108.653,397.817,-92.279,-178.623,15.587,150.992
C08963=1108.659,398.064,-92.317,-178.621,15.592,150.993
C08964=1108.665,398.312,-92.354,-178.619,15.597,150.994
C08965=1108.670,398.559,-92.392,-178.617,15.603,150.994
C08966=1108.676,398.806,-92.429,-178.614,15.608,150.995
C08967=1108.682,399.053,-92.467,-178.612,15.613,150.996
C08968=1108.687,399.299,-92.504,-178.610,15.618,150.997
C08969=1108.693,399.547,-92.541,-178.608,15.623,150.998
C08970=1108.698,399.794,-92.580,-178.606,15.629,150.999
C08971=1108.704,400.041,-92.618,-178.604,15.634,151.000
C08972=1108.710,400.288,-92.655,-178.602,15.639,151.000
C08973=1108.715,400.535,-92.693,-178.600,15.644,151.001
C08974=1108.721,400.782,-92.731,-178.597,15.649,151.002
C08975=1108.726,401.029,-92.768,-178.595,15.655,151.003
C08976=1108.732,401.276,-92.806,-178.593,15.660,151.004
C08977=1108.738,401.524,-92.844,-178.591,15.666,151.005
C08978=1108.744,401.771,-92.881,-178.589,15.671,151.006
C08979=1108.749,402.018,-92.920,-178.587,15.676,151.007
C08980=1108.755,402.265,-92.957,-178.585,15.682,151.008
C08981=1108.761,402.512,-92.995,-178.583,15.687,151.009
C08982=1108.766,402.759,-93.033,-178.581,15.692,151.009
C08983=1108.771,403.006,-93.071,-178.578,15.699,151.011
C08984=1108.777,403.253,-93.108,-178.576,15.704,151.011
C08985=1108.782,403.500,-93.147,-178.574,15.709,151.012
C08986=1108.788,403.747,-93.184,-178.572,15.715,151.013
C08987=1108.794,403.994,-93.223,-178.570,15.720,151.014
C08988=1108.800,404.241,-93.261,-178.568,15.726,151.015
C08989=1108.806,404.488,-93.299,-178.566,15.731,151.016
C08990=1108.811,404.735,-93.337,-178.564,15.737,151.017
C08991=1108.817,404.982,-93.375,-178.562,15.743,151.018
C08992=1108.822,405.229,-93.412,-178.560,15.749,151.019
C08993=1108.828,405.476,-93.450,-178.558,15.754,151.020
C08994=1108.834,405.724,-93.489,-178.556,15.760,151.021
C08995=1108.839,405.971,-93.527,-178.554,15.765,151.022
C08996=1108.845,406.218,-93.565,-178.552,15.772,151.023
C08997=1108.851,406.464,-93.603,-178.550,15.777,151.024
C08998=1108.856,406.711,-93.642,-178.548,15.783,151.025
C08999=1108.861,406.958,-93.680,-178.547,15.789,151.027
C09000=1108.868,407.205,-93.718,-178.545,15.794,151.028
C09001=1108.873,407.452,-93.757,-178.542,15.801,151.029
C09002=1108.879,407.699,-93.794,-178.540,15.806,151.030
C09003=1108.884,407.946,-93.833,-178.539,15.812,151.031
C09004=1108.889,408.193,-93.871,-178.536,15.818,151.032
C09005=1108.896,408.441,-93.909,-178.534,15.824,151.033
C09006=1108.901,408.688,-93.948,-178.533,15.830,151.034
C09007=1108.906,408.934,-93.987,-178.531,15.836,151.035
C09008=1108.912,409.181,-94.024,-178.529,15.842,151.036
C09009=1108.917,409.428,-94.063,-178.527,15.848,151.038
C09010=1108.923,409.676,-94.101,-178.525,15.854,151.039
C09011=1108.928,409.886,-94.135,-178.524,15.860,151.040
C09012=1108.933,410.099,-94.168,-178.522,15.865,151.041
C09013=1108.937,410.310,-94.200,-178.520,15.870,151.042
C09014=1108.942,410.522,-94.233,-178.519,15.876,151.043
C09015=1108.948,410.733,-94.266,-178.517,15.881,151.044
C09016=1108.952,410.945,-94.299,-178.516,15.886,151.045
C09017=1108.957,411.157,-94.332,-178.514,15.891,151.046
C09018=1108.962,411.369,-94.365,-178.512,15.896,151.047
C09019=1108.967,411.615,-94.404,-178.510,15.903,151.048
C09020=1108.972,411.862,-94.443,-178.509,15.909,151.049
C09021=1108.979,412.109,-94.481,-178.507,15.915,151.050
C09022=1108.984,412.356,-94.520,-178.505,15.922,151.052
C09023=1108.989,412.603,-94.558,-178.504,15.928,151.053
C09024=1108.995,412.850,-94.597,-178.501,15.935,151.054
C09025=1109.001,413.098,-94.636,-178.500,15.941,151.055
C09026=1109.006,413.344,-94.675,-178.498,15.948,151.056
C09027=1109.012,413.591,-94.713,-178.496,15.954,151.058
C09028=1109.018,413.838,-94.752,-178.494,15.960,151.059
C09029=1109.023,414.085,-94.790,-178.493,15.967,151.060
C09030=1109.029,414.331,-94.830,-178.490,15.973,151.062
C09031=1109.035,414.579,-94.868,-178.489,15.979,151.063
C09032=1109.040,414.826,-94.907,-178.487,15.987,151.064
C09033=1109.046,415.072,-94.946,-178.485,15.993,151.065
C09034=1109.052,415.319,-94.984,-178.484,16.000,151.067
C09035=1109.057,415.566,-95.024,-178.482,16.006,151.068
C09036=1109.063,415.813,-95.062,-178.480,16.013,151.069
C09037=1109.069,416.060,-95.101,-178.479,16.019,151.071
C09038=1109.074,416.306,-95.140,-178.477,16.026,151.072
C09039=1109.080,416.554,-95.179,-178.475,16.032,151.073
C09040=1109.085,416.801,-95.218,-178.473,16.039,151.075
C09041=1109.091,417.047,-95.257,-178.471,16.046,151.076
C09042=1109.097,417.294,-95.297,-178.470,16.053,151.078
C09043=1109.102,417.541,-95.335,-178.468,16.060,151.079
C09044=1109.108,417.788,-95.374,-178.467,16.066,151.080
C09045=1109.114,418.035,-95.414,-178.465,16.073,151.082
C09046=1109.119,418.281,-95.453,-178.463,16.080,151.083
C09047=1109.124,418.528,-95.491,-178.462,16.087,151.084
C09048=1109.130,418.775,-95.530,-178.460,16.094,151.086
C09049=1109.136,419.022,-95.569,-178.458,16.101,151.087
C09050=1109.141,419.269,-95.609,-178.457,16.108,151.089
C09051=1109.147,419.516,-95.649,-178.455,16.115,151.090
C09052=1109.152,419.762,-95.688,-178.454,16.123,151.092
C09053=1109.158,420.009,-95.727,-178.453,16.129,151.093
C09054=1109.164,420.256,-95.766,-178.451,16.137,151.095
C09055=1109.169,420.504,-95.805,-178.449,16.144,151.096
C09056=1109.175,420.750,-95.844,-178.447,16.151,151.098
C09057=1109.181,420.997,-95.883,-178.446,16.158,151.099
C09058=1109.186,421.244,-95.923,-178.445,16.165,151.101
C09059=1109.191,421.490,-95.962,-178.443,16.173,151.102
